KUKA KRL program: EPS_2_25694_SR01_A_NEW_20251202031151.src

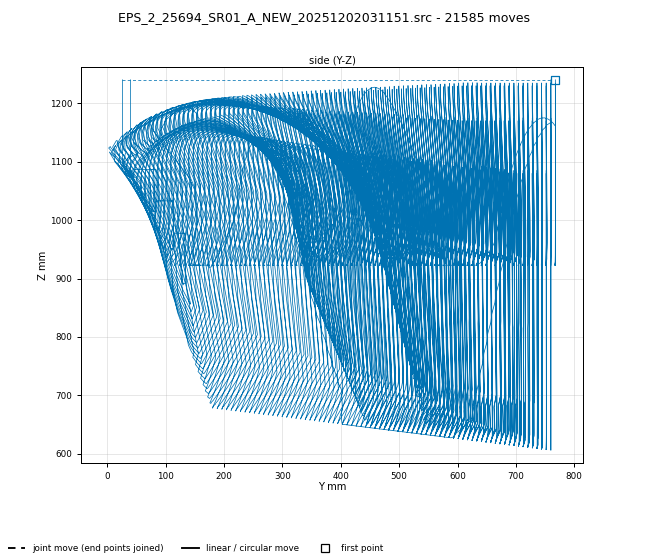
[picture p0: tool path of EPS_2_25694_SR01_A_NEW_20251202031151.src, 21585 of 21587 moves have a stored position in this frame; points joined in program order, loops and branches not executed]
&ACCESS RVP
&REL 4
&COMMENT QRS 19112012
&PARAM EDITMASK = *
DEF PART()
EXT BAS (BAS_COMMAND :IN,REAL :IN )
INT I
BAS (#INITMOV,0 )

;KUKA QRS Post kuka4.cps  Date:22-06-2017 !

File_ID=2935

QRS_PRE_INIT()

;Init var - Until changes are made in qrs_pre_init
Outlet_Square_prg=0
Inlet_1_Square_prg=0
Inlet_2_Square_prg=0
Inlet_3_Square_prg=0
Inlet_4_Square_prg=0
Inlet_5_Square_prg=0

Outlet_1={X 0.000, Y 612.000, Z 964.000, B 0.000, E1 0.000 }
Inlet_1={X 0.000, Y 612.000, Z 904.000, B 0.000, E1 90.000 }
Inlet_2={X 0.000, Y 692.870, Z 705.000, B 0.000, E1 260.000 }
Outlet_1_type=533
Inlet_1_type=533
Inlet_2_type=251
;QRS#1=Sidecore dimensions
;QRS#2=525-21" Concrete
;QRS#3=525-21" Concrete
;QRS#4=250-10" PVC SDR 35
;QRS#5=
;QRS#6=
;QRS#7=
;QRS#8=
;QRS#9=S306-32
;QRS#10=S306-32
;QRS#11=14M PSX
;QRS#12=
;QRS#13=
;QRS#14=
;QRS#15=
;QRS#16=1524x152x1676 5,5'
;QRS#17=EPS Height
;QRS#18=1230,5
;QRS#19=*
;QRS#20= UPDATED VERSION 22-06-2017
;QRS#21=*
Outlet_Square=0350
Inlet_1_Square=0350
Inlet_2_Square=0100
Inlet_3_Square=0
Inlet_4_Square=0
Inlet_5_Square=0
Mill_Square=1
Outlet_Square_Prg=263
Inlet_1_Square_prg=263
Inlet_2_Square_prg=205

QRS_INIT()

$ADVANCE=5

; T1
PTP {E1 173.088,E2 173.088}
PTP {X 0,Y 767.616,A -85,B 0,C 180,E1 173.088,E2 173.088,E3 0,E4 0,E5 0,E6 0}
QRS_SPEED_INIT()
LIN {X 0,Y 767.616,Z 1240.5,A -85,B 0,C 180,E1 173.088,E2 173.088,E3 0,E4 0,E5 0,E6 0} C_VEL
LIN {X 0,Y 767.616,Z 1171.13,A -85,B 0,C 180,E1 173.088,E2 173.088} C_VEL
LIN {X 0,Y 767.616,Z 1163.237,A -85,B 0,C 180,E1 173.088,E2 173.088} C_VEL
LIN {X 0,Y 767.6,Z 1161.315,A -85,B 0,C 180,E1 173.278,E2 173.278} C_VEL
LIN {X 0,Y 767.645,Z 1164.897,A -85,B 0,C 180,E1 174.209,E2 174.209} C_VEL
LIN {X 0,Y 767.804,Z 1167.383,A -85,B 0,C 180,E1 174.959,E2 174.959} C_VEL
LIN {X 0,Y 767.62,Z 1170.432,A -85,B 0,C 180,E1 176.081,E2 176.081} C_VEL
LIN {X 0,Y 767.646,Z 1172.644,A -85,B 0,C 180,E1 177.202,E2 177.202} C_VEL
LIN {X 0,Y 767.795,Z 1174.074,A -85,B 0,C 180,E1 178.323,E2 178.323} C_VEL
LIN {X 0,Y 767.585,Z 1174.722,A -85,B 0,C 180,E1 179.069,E2 179.069} C_VEL
LIN {X 0,Y 767.644,Z 1174.677,A -85,B 0,C 180,E1 180.934,E2 180.934} C_VEL
LIN {X 0,Y 767.742,Z 1173.598,A -85,B 0,C 180,E1 182.054,E2 182.054} C_VEL
LIN {X 0,Y 767.614,Z 1172.514,A -85,B 0,C 180,E1 182.801,E2 182.801} C_VEL
LIN {X 0,Y 767.666,Z 1170.222,A -85,B 0,C 180,E1 183.922,E2 183.922} C_VEL
LIN {X 0,Y 767.825,Z 1168.163,A -85,B 0,C 180,E1 184.669,E2 184.669} C_VEL
LIN {X 0,Y 767.693,Z 1165.832,A -85,B 0,C 180,E1 185.419,E2 185.419} C_VEL
LIN {X 0,Y 767.64,Z 1163.158,A -85,B 0,C 180,E1 186.17,E2 186.17} C_VEL
LIN {X 0,Y 767.709,Z 1160.308,A -85,B 0,C 180,E1 186.878,E2 186.878} C_VEL
LIN {X 0,Y 767.81,Z 1156.374,A -85,B 0,C 180,E1 187.718,E2 187.718} C_VEL
LIN {X 0,Y 767.635,Z 1150.131,A -85,B 0,C 180,E1 188.898,E2 188.898} C_VEL
LIN {X 0,Y 767.742,Z 1144.316,A -85,B 0,C 180,E1 189.842,E2 189.842} C_VEL
LIN {X 0,Y 767.829,Z 1139.474,A -85,B 0,C 180,E1 190.552,E2 190.552} C_VEL
LIN {X 0,Y 767.685,Z 1132.395,A -85,B 0,C 180,E1 191.504,E2 191.504} C_VEL
LIN {X 0,Y 767.755,Z 1123.331,A -85,B 0,C 180,E1 192.576,E2 192.576} C_VEL
LIN {X 0,Y 767.785,Z 1116.439,A -85,B 0,C 180,E1 193.319,E2 193.319} C_VEL
LIN {X 0,Y 767.704,Z 1107.11,A -85,B 0,C 180,E1 194.231,E2 194.231} C_VEL
LIN {X 0,Y 767.763,Z 1099.606,A -85,B 0,C 180,E1 194.904,E2 194.904} C_VEL
LIN {X 0,Y 767.79,Z 1090.202,A -85,B 0,C 180,E1 195.677,E2 195.677} C_VEL
LIN {X 0,Y 767.737,Z 1080.825,A -85,B 0,C 180,E1 196.385,E2 196.385} C_VEL
LIN {X 0,Y 767.747,Z 1071.416,A -85,B 0,C 180,E1 197.039,E2 197.039} C_VEL
LIN {X 0,Y 767.76,Z 1060.856,A -85,B 0,C 180,E1 197.71,E2 197.71} C_VEL
LIN {X 0,Y 767.758,Z 1050.335,A -85,B 0,C 180,E1 198.323,E2 198.323} C_VEL
LIN {X 0,Y 767.76,Z 1039.977,A -85,B 0,C 180,E1 198.877,E2 198.877} C_VEL
LIN {X 0,Y 767.736,Z 1028.552,A -85,B 0,C 180,E1 199.433,E2 199.433} C_VEL
LIN {X 0,Y 767.781,Z 1015.782,A -85,B 0,C 180,E1 199.989,E2 199.989} C_VEL
LIN {X 0,Y 767.752,Z 1003.711,A -85,B 0,C 180,E1 200.462,E2 200.462} C_VEL
LIN {X 0,Y 767.714,Z 992.2,A -85,B 0,C 180,E1 200.866,E2 200.866} C_VEL
LIN {X 0,Y 767.776,Z 978.277,A -85,B 0,C 180,E1 201.291,E2 201.291} C_VEL
LIN {X 0,Y 767.685,Z 965.195,A -85,B 0,C 180,E1 201.639,E2 201.639} C_VEL
LIN {X 0,Y 767.732,Z 952.435,A -85,B 0,C 180,E1 201.925,E2 201.925} C_VEL
LIN {X 0,Y 767.714,Z 939.22,A -85,B 0,C 180,E1 202.172,E2 202.172} C_VEL
LIN {X 0,Y 767.488,Z 929.301,A -85,B 0,C 180,E1 202.333,E2 202.333} C_VEL
LIN {X 0,Y 766.705,Z 923.03,A -85,B 0,C 180,E1 202.439,E2 202.439} C_VEL
LIN {X 0,Y 767.325,Z 923.03,A -85,B 0,C 180,E1 202.504,E2 202.504} C_VEL
LIN {X 0,Y 767.822,Z 923.03,A -85,B 0,C 180,E1 202.614,E2 202.614} C_VEL
LIN {X 0,Y 767.644,Z 923.03,A -85,B 0,C 180,E1 203.63,E2 203.63} C_VEL
LIN {X 0,Y 767.743,Z 923.03,A -85,B 0,C 180,E1 208.169,E2 208.169} C_VEL
LIN {X 0,Y 767.312,Z 923.03,A -85,B 0,C 180,E1 210.325,E2 210.325} C_VEL
LIN {X 0,Y 767.713,Z 923.03,A -85,B 0,C 180,E1 212.493,E2 212.493} C_VEL
LIN {X 0,Y 767.395,Z 923.03,A -85,B 0,C 180,E1 213.845,E2 213.845} C_VEL
LIN {X 0,Y 767.696,Z 923.03,A -85,B 0,C 180,E1 217.093,E2 217.093} C_VEL
LIN {X 0,Y 767.102,Z 923.03,A -85,B 0,C 180,E1 220.031,E2 220.031} C_VEL
LIN {X 0,Y 767.566,Z 923.03,A -85,B 0,C 180,E1 221.878,E2 221.878} C_VEL
LIN {X 0,Y 767.622,Z 923.03,A -85,B 0,C 180,E1 222.894,E2 222.894} C_VEL
LIN {X 0,Y 767.591,Z 923.03,A -85,B 0,C 180,E1 227.109,E2 227.109} C_VEL
LIN {X 0,Y 767.541,Z 923.03,A -85,B 0,C 180,E1 228.12,E2 228.12} C_VEL
LIN {X 0,Y 767.131,Z 923.03,A -85,B 0,C 180,E1 230.554,E2 230.554} C_VEL
LIN {X 0,Y 767.736,Z 923.03,A -85,B 0,C 180,E1 232.966,E2 232.966} C_VEL
LIN {X 0,Y 767.601,Z 923.03,A -85,B 0,C 180,E1 236.132,E2 236.132} C_VEL
LIN {X 0,Y 767.507,Z 923.03,A -85,B 0,C 180,E1 237.497,E2 237.497} C_VEL
LIN {X 0,Y 767.223,Z 923.03,A -85,B 0,C 180,E1 239.69,E2 239.69} C_VEL
LIN {X 0,Y 767.749,Z 923.03,A -85,B 0,C 180,E1 241.832,E2 241.832} C_VEL
LIN {X 0,Y 767.82,Z 923.03,A -85,B 0,C 180,E1 246.871,E2 246.871} C_VEL
LIN {X 0,Y 767.647,Z 923.03,A -85,B 0,C 180,E1 246.92,E2 246.92} C_VEL
LIN {X 0,Y 767.578,Z 923.795,A -85,B 0,C 180,E1 246.945,E2 246.945} C_VEL
LIN {X 0,Y 767.629,Z 977.672,A -85,B 0,C 180,E1 247.486,E2 247.486} C_VEL
LIN {X 0,Y 767.739,Z 990.959,A -85,B 0,C 180,E1 247.656,E2 247.656} C_VEL
LIN {X 0,Y 767.675,Z 1003.622,A -85,B 0,C 180,E1 247.858,E2 247.858} C_VEL
LIN {X 0,Y 767.717,Z 1014.508,A -85,B 0,C 180,E1 248.07,E2 248.07} C_VEL
LIN {X 0,Y 767.776,Z 1030.265,A -85,B 0,C 180,E1 248.446,E2 248.446} C_VEL
LIN {X 0,Y 767.72,Z 1042.52,A -85,B 0,C 180,E1 248.785,E2 248.785} C_VEL
LIN {X 0,Y 767.741,Z 1055.126,A -85,B 0,C 180,E1 249.188,E2 249.188} C_VEL
LIN {X 0,Y 767.772,Z 1067.885,A -85,B 0,C 180,E1 249.651,E2 249.651} C_VEL
LIN {X 0,Y 767.73,Z 1079.832,A -85,B 0,C 180,E1 250.134,E2 250.134} C_VEL
LIN {X 0,Y 767.776,Z 1092.122,A -85,B 0,C 180,E1 250.692,E2 250.692} C_VEL
LIN {X 0,Y 767.784,Z 1103.222,A -85,B 0,C 180,E1 251.247,E2 251.247} C_VEL
LIN {X 0,Y 767.77,Z 1114.39,A -85,B 0,C 180,E1 251.862,E2 251.862} C_VEL
LIN {X 0,Y 767.759,Z 1124.576,A -85,B 0,C 180,E1 252.474,E2 252.474} C_VEL
LIN {X 0,Y 767.741,Z 1133.933,A -85,B 0,C 180,E1 253.083,E2 253.083} C_VEL
LIN {X 0,Y 767.808,Z 1144.001,A -85,B 0,C 180,E1 253.803,E2 253.803} C_VEL
LIN {X 0,Y 767.769,Z 1153.202,A -85,B 0,C 180,E1 254.517,E2 254.517} C_VEL
LIN {X 0,Y 767.702,Z 1162.313,A -85,B 0,C 180,E1 255.288,E2 255.288} C_VEL
LIN {X 0,Y 767.775,Z 1170.487,A -85,B 0,C 180,E1 256.045,E2 256.045} C_VEL
LIN {X 0,Y 767.79,Z 1178.25,A -85,B 0,C 180,E1 256.827,E2 256.827} C_VEL
LIN {X 0,Y 767.68,Z 1185.844,A -85,B 0,C 180,E1 257.662,E2 257.662} C_VEL
LIN {X 0,Y 767.726,Z 1192.732,A -85,B 0,C 180,E1 258.497,E2 258.497} C_VEL
LIN {X 0,Y 767.83,Z 1198.109,A -85,B 0,C 180,E1 259.211,E2 259.211} C_VEL
LIN {X 0,Y 767.639,Z 1204.639,A -85,B 0,C 180,E1 260.157,E2 260.157} C_VEL
LIN {X 0,Y 767.667,Z 1210.401,A -85,B 0,C 180,E1 261.102,E2 261.102} C_VEL
LIN {X 0,Y 767.825,Z 1215.453,A -85,B 0,C 180,E1 262.047,E2 262.047} C_VEL
LIN {X 0,Y 767.632,Z 1221.05,A -85,B 0,C 180,E1 263.258,E2 263.258} C_VEL
LIN {X 0,Y 767.708,Z 1224.727,A -85,B 0,C 180,E1 264.206,E2 264.206} C_VEL
LIN {X 0,Y 767.823,Z 1227.22,A -85,B 0,C 180,E1 264.957,E2 264.957} C_VEL
LIN {X 0,Y 767.655,Z 1229.333,A -85,B 0,C 180,E1 265.704,E2 265.704} C_VEL
LIN {X 0,Y 767.605,Z 1231.115,A -85,B 0,C 180,E1 266.452,E2 266.452} C_VEL
LIN {X 0,Y 767.683,Z 1232.567,A -85,B 0,C 180,E1 267.2,E2 267.2} C_VEL
LIN {X 0,Y 767.835,Z 1233.648,A -85,B 0,C 180,E1 267.947,E2 267.947} C_VEL
LIN {X 0,Y 767.616,Z 1234.703,A -85,B 0,C 180,E1 269.066,E2 269.066} C_VEL
LIN {X 0,Y 767.835,Z 1234.661,A -85,B 0,C 180,E1 270.931,E2 270.931} C_VEL
LIN {X 0,Y 767.781,Z 1234.037,A -85,B 0,C 180,E1 271.678,E2 271.678} C_VEL
LIN {X 0,Y 767.801,Z 1232.548,A -85,B 0,C 180,E1 272.798,E2 272.798} C_VEL
LIN {X 0,Y 767.672,Z 1231.107,A -85,B 0,C 180,E1 273.545,E2 273.545} C_VEL
LIN {X 0,Y 767.7,Z 1228.315,A -85,B 0,C 180,E1 274.667,E2 274.667} C_VEL
LIN {X 0,Y 767.838,Z 1225.965,A -85,B 0,C 180,E1 275.415,E2 275.415} C_VEL
LIN {X 0,Y 767.7,Z 1223.339,A -85,B 0,C 180,E1 276.166,E2 276.166} C_VEL
LIN {X 0,Y 767.635,Z 1220.661,A -85,B 0,C 180,E1 276.839,E2 276.839} C_VEL
LIN {X 0,Y 767.801,Z 1215.469,A -85,B 0,C 180,E1 277.951,E2 277.951} C_VEL
LIN {X 0,Y 767.723,Z 1210.407,A -85,B 0,C 180,E1 278.895,E2 278.895} C_VEL
LIN {X 0,Y 767.638,Z 1204.655,A -85,B 0,C 180,E1 279.841,E2 279.841} C_VEL
LIN {X 0,Y 767.786,Z 1198.133,A -85,B 0,C 180,E1 280.787,E2 280.787} C_VEL
LIN {X 0,Y 767.73,Z 1190.839,A -85,B 0,C 180,E1 281.739,E2 281.739} C_VEL
LIN {X 0,Y 767.66,Z 1183.778,A -85,B 0,C 180,E1 282.575,E2 282.575} C_VEL
LIN {X 0,Y 767.78,Z 1175.272,A -85,B 0,C 180,E1 283.479,E2 283.479} C_VEL
LIN {X 0,Y 767.762,Z 1167.631,A -85,B 0,C 180,E1 284.227,E2 284.227} C_VEL
LIN {X 0,Y 767.71,Z 1159.021,A -85,B 0,C 180,E1 284.999,E2 284.999} C_VEL
LIN {X 0,Y 767.753,Z 1150.824,A -85,B 0,C 180,E1 285.675,E2 285.675} C_VEL
LIN {X 0,Y 767.789,Z 1141.234,A -85,B 0,C 180,E1 286.4,E2 286.4} C_VEL
LIN {X 0,Y 767.753,Z 1132.152,A -85,B 0,C 180,E1 287.036,E2 287.036} C_VEL
LIN {X 0,Y 767.756,Z 1120.627,A -85,B 0,C 180,E1 287.769,E2 287.769} C_VEL
LIN {X 0,Y 767.748,Z 1110.08,A -85,B 0,C 180,E1 288.382,E2 288.382} C_VEL
LIN {X 0,Y 767.777,Z 1099.692,A -85,B 0,C 180,E1 288.935,E2 288.935} C_VEL
LIN {X 0,Y 767.775,Z 1088.232,A -85,B 0,C 180,E1 289.491,E2 289.491} C_VEL
LIN {X 0,Y 767.732,Z 1076.974,A -85,B 0,C 180,E1 289.987,E2 289.987} C_VEL
LIN {X 0,Y 767.792,Z 1064.346,A -85,B 0,C 180,E1 290.483,E2 290.483} C_VEL
LIN {X 0,Y 767.771,Z 1051.74,A -85,B 0,C 180,E1 290.924,E2 290.924} C_VEL
LIN {X 0,Y 767.668,Z 1038.39,A -85,B 0,C 180,E1 291.336,E2 291.336} C_VEL
LIN {X 0,Y 767.771,Z 1025.24,A -85,B 0,C 180,E1 291.68,E2 291.68} C_VEL
LIN {X 0,Y 767.797,Z 1012.208,A -85,B 0,C 180,E1 291.972,E2 291.972} C_VEL
LIN {X 0,Y 767.692,Z 999.283,A -85,B 0,C 180,E1 292.216,E2 292.216} C_VEL
LIN {X 0,Y 767.662,Z 989.615,A -85,B 0,C 180,E1 292.367,E2 292.367} C_VEL
LIN {X 0,Y 767.711,Z 970.479,A -85,B 0,C 180,E1 292.587,E2 292.587} C_VEL
LIN {X 0,Y 767.567,Z 923.965,A -85,B 0,C 180,E1 293.054,E2 293.054} C_VEL
LIN {X 0,Y 767.609,Z 923.03,A -85,B 0,C 180,E1 293.072,E2 293.072} C_VEL
LIN {X 0,Y 767.756,Z 923.03,A -85,B 0,C 180,E1 293.108,E2 293.108} C_VEL
LIN {X 0,Y 767.439,Z 923.03,A -85,B 0,C 180,E1 294.021,E2 294.021} C_VEL
LIN {X 0,Y 767.75,Z 923.03,A -85,B 0,C 180,E1 298.166,E2 298.166} C_VEL
LIN {X 0,Y 767.337,Z 923.03,A -85,B 0,C 180,E1 300.324,E2 300.324} C_VEL
LIN {X 0,Y 767.758,Z 923.03,A -85,B 0,C 180,E1 302.488,E2 302.488} C_VEL
LIN {X 0,Y 767.431,Z 923.03,A -85,B 0,C 180,E1 303.849,E2 303.849} C_VEL
LIN {X 0,Y 767.734,Z 923.03,A -85,B 0,C 180,E1 307.096,E2 307.096} C_VEL
LIN {X 0,Y 767.112,Z 923.03,A -85,B 0,C 180,E1 310.032,E2 310.032} C_VEL
LIN {X 0,Y 767.566,Z 923.03,A -85,B 0,C 180,E1 311.875,E2 311.875} C_VEL
LIN {X 0,Y 767.634,Z 923.03,A -85,B 0,C 180,E1 312.895,E2 312.895} C_VEL
LIN {X 0,Y 767.633,Z 923.03,A -85,B 0,C 180,E1 317.102,E2 317.102} C_VEL
LIN {X 0,Y 767.581,Z 923.03,A -85,B 0,C 180,E1 318.123,E2 318.123} C_VEL
LIN {X 0,Y 767.123,Z 923.03,A -85,B 0,C 180,E1 320.554,E2 320.554} C_VEL
LIN {X 0,Y 767.7,Z 923.03,A -85,B 0,C 180,E1 322.964,E2 322.964} C_VEL
LIN {X 0,Y 767.576,Z 923.03,A -85,B 0,C 180,E1 326.13,E2 326.13} C_VEL
LIN {X 0,Y 767.481,Z 923.03,A -85,B 0,C 180,E1 327.496,E2 327.496} C_VEL
LIN {X 0,Y 767.213,Z 923.03,A -85,B 0,C 180,E1 329.687,E2 329.687} C_VEL
LIN {X 0,Y 767.767,Z 923.03,A -85,B 0,C 180,E1 331.832,E2 331.832} C_VEL
LIN {X 0,Y 767.786,Z 923.03,A -85,B 0,C 180,E1 335.988,E2 335.988} C_VEL
LIN {X 0,Y 767.774,Z 923.03,A -85,B 0,C 180,E1 340.011,E2 340.011} C_VEL
LIN {X 0,Y 767.215,Z 923.03,A -85,B 0,C 180,E1 343.947,E2 343.947} C_VEL
LIN {X 0,Y 767.659,Z 923.03,A -85,B 0,C 180,E1 345.865,E2 345.865} C_VEL
LIN {X 0,Y 767.793,Z 923.03,A -85,B 0,C 180,E1 349.685,E2 349.685} C_VEL
LIN {X 0,Y 767.822,Z 923.03,A -85,B 0,C 180,E1 353.457,E2 353.457} C_VEL
LIN {X 0,Y 767.841,Z 923.03,A -85,B 0,C 180,E1 357.918,E2 357.918} C_VEL
LIN {X 0,Y 767.412,Z 923.03,A -85,B 0,C 180,E1 358.035,E2 358.035} C_VEL
LIN {X 0,Y 766.897,Z 923.03,A -85,B 0,C 180,E1 358.098,E2 358.098} C_VEL
LIN {X 0,Y 767.682,Z 928.435,A -85,B 0,C 180,E1 358.165,E2 358.165} C_VEL
LIN {X 0,Y 767.803,Z 954.739,A -85,B 0,C 180,E1 358.423,E2 358.423} C_VEL
LIN {X 0,Y 767.86,Z 965.313,A -85,B 0,C 180,E1 358.583,E2 358.583} C_VEL
LIN {X 0,Y 767.858,Z 973.85,A -85,B 0,C 180,E1 358.755,E2 358.755} C_VEL
LIN {X 0,Y 767.845,Z 982.97,A -85,B 0,C 180,E1 358.98,E2 358.98} C_VEL
LIN {X 0,Y 767.836,Z 991.896,A -85,B 0,C 180,E1 359.253,E2 359.253} C_VEL
LIN {X 0,Y 767.828,Z 999.738,A -85,B 0,C 180,E1 359.532,E2 359.532} C_VEL
LIN {X 0,Y 767.806,Z 1008.817,A -85,B 0,C 180,E1 359.905,E2 359.905} C_VEL
LIN {X 0,Y 767.817,Z 1016.57,A -85,B 0,C 180,E1 360.278,E2 360.278} C_VEL
LIN {X 0,Y 767.843,Z 1023.443,A -85,B 0,C 180,E1 360.651,E2 360.651} C_VEL
LIN {X 0,Y 767.856,Z 1031.11,A -85,B 0,C 180,E1 361.118,E2 361.118} C_VEL
LIN {X 0,Y 767.816,Z 1037.833,A -85,B 0,C 180,E1 361.584,E2 361.584} C_VEL
LIN {X 0,Y 767.828,Z 1046.128,A -85,B 0,C 180,E1 362.237,E2 362.237} C_VEL
LIN {X 0,Y 767.834,Z 1052.24,A -85,B 0,C 180,E1 362.797,E2 362.797} C_VEL
LIN {X 0,Y 767.79,Z 1057.697,A -85,B 0,C 180,E1 363.358,E2 363.358} C_VEL
LIN {X 0,Y 767.808,Z 1062.52,A -85,B 0,C 180,E1 363.918,E2 363.918} C_VEL
LIN {X 0,Y 767.858,Z 1066.717,A -85,B 0,C 180,E1 364.479,E2 364.479} C_VEL
LIN {X 0,Y 767.776,Z 1070.444,A -85,B 0,C 180,E1 365.041,E2 365.041} C_VEL
LIN {X 0,Y 767.747,Z 1073.688,A -85,B 0,C 180,E1 365.603,E2 365.603} C_VEL
LIN {X 0,Y 767.808,Z 1076.465,A -85,B 0,C 180,E1 366.165,E2 366.165} C_VEL
LIN {X 0,Y 767.817,Z 1079.418,A -85,B 0,C 180,E1 366.877,E2 366.877} C_VEL
LIN {X 0,Y 767.756,Z 1081.384,A -85,B 0,C 180,E1 367.481,E2 367.481} C_VEL
LIN {X 0,Y 767.762,Z 1082.621,A -85,B 0,C 180,E1 367.951,E2 367.951} C_VEL
LIN {X 0,Y 767.82,Z 1083.578,A -85,B 0,C 180,E1 368.422,E2 368.422} C_VEL
LIN {X 0,Y 767.773,Z 1084.727,A -85,B 0,C 180,E1 369.366,E2 369.366} C_VEL
LIN {X 0,Y 767.751,Z 1084.916,A -85,B 0,C 180,E1 369.839,E2 369.839} C_VEL
LIN {X 0,Y 767.782,Z 1084.839,A -85,B 0,C 180,E1 370.312,E2 370.312} C_VEL
LIN {X 0,Y 767.852,Z 1084.497,A -85,B 0,C 180,E1 370.786,E2 370.786} C_VEL
LIN {X 0,Y 767.8,Z 1083.921,A -85,B 0,C 180,E1 371.262,E2 371.262} C_VEL
LIN {X 0,Y 767.746,Z 1083.082,A -85,B 0,C 180,E1 371.738,E2 371.738} C_VEL
LIN {X 0,Y 767.744,Z 1081.966,A -85,B 0,C 180,E1 372.215,E2 372.215} C_VEL
LIN {X 0,Y 767.795,Z 1080.566,A -85,B 0,C 180,E1 372.692,E2 372.692} C_VEL
LIN {X 0,Y 767.787,Z 1077.674,A -85,B 0,C 180,E1 373.474,E2 373.474} C_VEL
LIN {X 0,Y 767.765,Z 1074.632,A -85,B 0,C 180,E1 374.13,E2 374.13} C_VEL
LIN {X 0,Y 767.803,Z 1071.423,A -85,B 0,C 180,E1 374.707,E2 374.707} C_VEL
LIN {X 0,Y 767.831,Z 1067.715,A -85,B 0,C 180,E1 375.286,E2 375.286} C_VEL
LIN {X 0,Y 767.772,Z 1063.48,A -85,B 0,C 180,E1 375.868,E2 375.868} C_VEL
LIN {X 0,Y 767.817,Z 1057.741,A -85,B 0,C 180,E1 376.547,E2 376.547} C_VEL
LIN {X 0,Y 767.845,Z 1051.803,A -85,B 0,C 180,E1 377.155,E2 377.155} C_VEL
LIN {X 0,Y 767.798,Z 1044.974,A -85,B 0,C 180,E1 377.767,E2 377.767} C_VEL
LIN {X 0,Y 767.836,Z 1037.134,A -85,B 0,C 180,E1 378.379,E2 378.379} C_VEL
LIN {X 0,Y 767.851,Z 1029.859,A -85,B 0,C 180,E1 378.871,E2 378.871} C_VEL
LIN {X 0,Y 767.826,Z 1022.668,A -85,B 0,C 180,E1 379.303,E2 379.303} C_VEL
LIN {X 0,Y 767.83,Z 1014.515,A -85,B 0,C 180,E1 379.736,E2 379.736} C_VEL
LIN {X 0,Y 767.84,Z 1006.03,A -85,B 0,C 180,E1 380.123,E2 380.123} C_VEL
LIN {X 0,Y 767.833,Z 997.385,A -85,B 0,C 180,E1 380.467,E2 380.467} C_VEL
LIN {X 0,Y 767.802,Z 988.868,A -85,B 0,C 180,E1 380.756,E2 380.756} C_VEL
LIN {X 0,Y 767.856,Z 979.688,A -85,B 0,C 180,E1 381.014,E2 381.014} C_VEL
LIN {X 0,Y 767.86,Z 969.785,A -85,B 0,C 180,E1 381.244,E2 381.244} C_VEL
LIN {X 0,Y 767.815,Z 959.779,A -85,B 0,C 180,E1 381.417,E2 381.417} C_VEL
LIN {X 0,Y 767.834,Z 950.7,A -85,B 0,C 180,E1 381.532,E2 381.532} C_VEL
LIN {X 0,Y 767.761,Z 926.079,A -85,B 0,C 180,E1 381.766,E2 381.766} C_VEL
LIN {X 0,Y 766.941,Z 923.622,A -85,B 0,C 180,E1 381.802,E2 381.802} C_VEL
LIN {X 0,Y 766.65,Z 923.03,A -85,B 0,C 180,E1 381.819,E2 381.819} C_VEL
LIN {X 0,Y 767.601,Z 923.03,A -85,B 0,C 180,E1 381.989,E2 381.989} C_VEL
LIN {X 0,Y 767.531,Z 923.03,A -85,B 0,C 180,E1 384.018,E2 384.018} C_VEL
LIN {X 0,Y 767.633,Z 923.03,A -85,B 0,C 180,E1 386.074,E2 386.074} C_VEL
LIN {X 0,Y 767.775,Z 923.03,A -85,B 0,C 180,E1 390.385,E2 390.385} C_VEL
LIN {X 0,Y 767.726,Z 923.03,A -85,B 0,C 180,E1 394.729,E2 394.729} C_VEL
LIN {X 0,Y 767.234,Z 923.03,A -85,B 0,C 180,E1 397.059,E2 397.059} C_VEL
LIN {X 0,Y 767.688,Z 923.03,A -85,B 0,C 180,E1 399.408,E2 399.408} C_VEL
LIN {X 0,Y 767.67,Z 923.03,A -85,B 0,C 180,E1 400.085,E2 400.085} C_VEL
LIN {X 0,Y 767.475,Z 923.03,A -85,B 0,C 180,E1 404.439,E2 404.439} C_VEL
LIN {X 0,Y 767.642,Z 923.03,A -85,B 0,C 180,E1 405.573,E2 405.573} C_VEL
LIN {X 0,Y 767.693,Z 923.03,A -85,B 0,C 180,E1 409.912,E2 409.912} C_VEL
LIN {X 0,Y 767.697,Z 923.03,A -85,B 0,C 180,E1 410.592,E2 410.592} C_VEL
LIN {X 0,Y 767.21,Z 923.03,A -85,B 0,C 180,E1 412.951,E2 412.951} C_VEL
LIN {X 0,Y 767.666,Z 923.03,A -85,B 0,C 180,E1 415.267,E2 415.267} C_VEL
LIN {X 0,Y 767.73,Z 923.03,A -85,B 0,C 180,E1 419.62,E2 419.62} C_VEL
LIN {X 0,Y 767.786,Z 923.03,A -85,B 0,C 180,E1 423.531,E2 423.531} C_VEL
LIN {X 0,Y 767.789,Z 923.03,A -85,B 0,C 180,E1 423.932,E2 423.932} C_VEL
LIN {X 0,Y 767.77,Z 923.03,A -85,B 0,C 180,E1 428.016,E2 428.016} C_VEL
LIN {X 0,Y 767.757,Z 923.03,A -85,B 0,C 180,E1 431.986,E2 431.986} C_VEL
LIN {X 0,Y 767.458,Z 923.03,A -85,B 0,C 180,E1 433.931,E2 433.931} C_VEL
LIN {X 0,Y 767.591,Z 923.03,A -85,B 0,C 180,E1 435.866,E2 435.866} C_VEL
LIN {X 0,Y 767.792,Z 923.03,A -85,B 0,C 180,E1 439.687,E2 439.687} C_VEL
LIN {X 0,Y 767.847,Z 923.03,A -85,B 0,C 180,E1 443.459,E2 443.459} C_VEL
LIN {X 0,Y 767.872,Z 923.03,A -85,B 0,C 180,E1 447.203,E2 447.203} C_VEL
LIN {X 0,Y 767.868,Z 923.03,A -85,B 0,C 180,E1 450.934,E2 450.934} C_VEL
LIN {X 0,Y 767.84,Z 923.03,A -85,B 0,C 180,E1 454.669,E2 454.669} C_VEL
LIN {X 0,Y 767.829,Z 923.03,A -85,B 0,C 180,E1 458.424,E2 458.424} C_VEL
LIN {X 0,Y 767.822,Z 923.03,A -85,B 0,C 180,E1 462.216,E2 462.216} C_VEL
LIN {X 0,Y 767.858,Z 923.03,A -85,B 0,C 180,E1 466.221,E2 466.221} C_VEL
LIN {X 0,Y 767.739,Z 923.03,A -85,B 0,C 180,E1 469.989,E2 469.989} C_VEL
LIN {X 0,Y 767.734,Z 923.03,A -85,B 0,C 180,E1 474.014,E2 474.014} C_VEL
LIN {X 0,Y 767.335,Z 923.03,A -85,B 0,C 180,E1 476.401,E2 476.401} C_VEL
LIN {X 0,Y 767.741,Z 923.03,A -85,B 0,C 180,E1 478.168,E2 478.168} C_VEL
LIN {X 0,Y 767.316,Z 923.03,A -85,B 0,C 180,E1 480.328,E2 480.328} C_VEL
LIN {X 0,Y 767.737,Z 923.03,A -85,B 0,C 180,E1 482.492,E2 482.492} C_VEL
LIN {X 0,Y 767.415,Z 923.03,A -85,B 0,C 180,E1 483.853,E2 483.853} C_VEL
LIN {X 0,Y 767.681,Z 923.03,A -85,B 0,C 180,E1 487.096,E2 487.096} C_VEL
LIN {X 0,Y 767.162,Z 923.03,A -85,B 0,C 180,E1 490.041,E2 490.041} C_VEL
LIN {X 0,Y 767.682,Z 923.03,A -85,B 0,C 180,E1 491.87,E2 491.87} C_VEL
LIN {X 0,Y 767.693,Z 923.03,A -85,B 0,C 180,E1 492.904,E2 492.904} C_VEL
LIN {X 0,Y 767.672,Z 923.03,A -85,B 0,C 180,E1 494.428,E2 494.428} C_VEL
LIN {X 0,Y 767.629,Z 923.03,A -85,B 0,C 180,E1 495.573,E2 495.573} C_VEL
LIN {X 0,Y 767.694,Z 923.03,A -85,B 0,C 180,E1 499.916,E2 499.916} C_VEL
LIN {X 0,Y 767.699,Z 923.03,A -85,B 0,C 180,E1 500.593,E2 500.593} C_VEL
LIN {X 0,Y 767.207,Z 923.03,A -85,B 0,C 180,E1 502.956,E2 502.956} C_VEL
LIN {X 0,Y 767.69,Z 923.03,A -85,B 0,C 180,E1 505.269,E2 505.269} C_VEL
LIN {X 0,Y 767.733,Z 923.03,A -85,B 0,C 180,E1 509.625,E2 509.625} C_VEL
LIN {X 0,Y 767.776,Z 923.03,A -85,B 0,C 180,E1 513.539,E2 513.539} C_VEL
LIN {X 0,Y 767.785,Z 923.03,A -85,B 0,C 180,E1 513.932,E2 513.932} C_VEL
LIN {X 0,Y 767.701,Z 923.03,A -85,B 0,C 180,E1 516.902,E2 516.902} C_VEL
LIN {X 0,Y 767.753,Z 923.03,A -85,B 0,C 180,E1 517.407,E2 517.407} C_VEL
LIN {X 0,Y 767.323,Z 923.03,A -85,B 0,C 180,E1 517.489,E2 517.489} C_VEL
LIN {X 0,Y 767.582,Z 936.224,A -85,B 0,C 180,E1 517.688,E2 517.688} C_VEL
LIN {X 0,Y 767.747,Z 945.654,A -85,B 0,C 180,E1 517.854,E2 517.854} C_VEL
LIN {X 0,Y 767.798,Z 957.639,A -85,B 0,C 180,E1 518.099,E2 518.099} C_VEL
LIN {X 0,Y 767.761,Z 969.731,A -85,B 0,C 180,E1 518.386,E2 518.386} C_VEL
LIN {X 0,Y 767.673,Z 980.092,A -85,B 0,C 180,E1 518.666,E2 518.666} C_VEL
LIN {X 0,Y 767.749,Z 995.086,A -85,B 0,C 180,E1 519.141,E2 519.141} C_VEL
LIN {X 0,Y 767.699,Z 1008.532,A -85,B 0,C 180,E1 519.629,E2 519.629} C_VEL
LIN {X 0,Y 767.775,Z 1019.516,A -85,B 0,C 180,E1 520.076,E2 520.076} C_VEL
LIN {X 0,Y 767.782,Z 1031.84,A -85,B 0,C 180,E1 520.634,E2 520.634} C_VEL
LIN {X 0,Y 767.731,Z 1042.97,A -85,B 0,C 180,E1 521.187,E2 521.187} C_VEL
LIN {X 0,Y 767.771,Z 1054.163,A -85,B 0,C 180,E1 521.803,E2 521.803} C_VEL
LIN {X 0,Y 767.779,Z 1065.314,A -85,B 0,C 180,E1 522.477,E2 522.477} C_VEL
LIN {X 0,Y 767.803,Z 1074.61,A -85,B 0,C 180,E1 523.088,E2 523.088} C_VEL
LIN {X 0,Y 767.75,Z 1084.792,A -85,B 0,C 180,E1 523.817,E2 523.817} C_VEL
LIN {X 0,Y 767.741,Z 1093.775,A -85,B 0,C 180,E1 524.519,E2 524.519} C_VEL
LIN {X 0,Y 767.824,Z 1101.772,A -85,B 0,C 180,E1 525.197,E2 525.197} C_VEL
LIN {X 0,Y 767.822,Z 1110.849,A -85,B 0,C 180,E1 526.037,E2 526.037} C_VEL
LIN {X 0,Y 767.788,Z 1118.688,A -85,B 0,C 180,E1 526.83,E2 526.83} C_VEL
LIN {X 0,Y 767.684,Z 1126.242,A -85,B 0,C 180,E1 527.665,E2 527.665} C_VEL
LIN {X 0,Y 767.739,Z 1133.09,A -85,B 0,C 180,E1 528.5,E2 528.5} C_VEL
LIN {X 0,Y 767.847,Z 1138.468,A -85,B 0,C 180,E1 529.214,E2 529.214} C_VEL
LIN {X 0,Y 767.649,Z 1144.953,A -85,B 0,C 180,E1 530.159,E2 530.159} C_VEL
LIN {X 0,Y 767.67,Z 1150.678,A -85,B 0,C 180,E1 531.105,E2 531.105} C_VEL
LIN {X 0,Y 767.82,Z 1155.701,A -85,B 0,C 180,E1 532.049,E2 532.049} C_VEL
LIN {X 0,Y 767.592,Z 1160.956,A -85,B 0,C 180,E1 533.188,E2 533.188} C_VEL
LIN {X 0,Y 767.6,Z 1161.315,A -85,B 0,C 180,E1 533.278,E2 533.278} C_VEL
LIN {X 0,Y 763.716,Z 1166.407,A -85,B 0,C 180,E1 534.508,E2 534.508} C_VEL
LIN {X 0,Y 759.772,Z 1170.193,A -85,B 0,C 180,E1 535.763,E2 535.763} C_VEL
LIN {X 0,Y 759.753,Z 1175.122,A -85,B 0,C 180,E1 538.859,E2 538.859} C_VEL
LIN {X 0,Y 759.763,Z 1175.045,A -85,B 0,C 180,E1 541.138,E2 541.138} C_VEL
LIN {X 0,Y 759.796,Z 1170.633,A -85,B 0,C 180,E1 543.99,E2 543.99} C_VEL
LIN {X 0,Y 759.882,Z 1159.817,A -85,B 0,C 180,E1 547.138,E2 547.138} C_VEL
LIN {X 0,Y 759.896,Z 1144.053,A -85,B 0,C 180,E1 550.019,E2 550.019} C_VEL
LIN {X 0,Y 759.952,Z 1123.015,A -85,B 0,C 180,E1 552.753,E2 552.753} C_VEL
LIN {X 0,Y 760.002,Z 1097.093,A -85,B 0,C 180,E1 555.273,E2 555.273} C_VEL
LIN {X 0,Y 760.101,Z 1066.649,A -85,B 0,C 180,E1 557.528,E2 557.528} C_VEL
LIN {X 0,Y 760.175,Z 1032.454,A -85,B 0,C 180,E1 559.447,E2 559.447} C_VEL
LIN {X 0,Y 760.291,Z 993.537,A -85,B 0,C 180,E1 561.037,E2 561.037} C_VEL
LIN {X 0,Y 760.392,Z 952.645,A -85,B 0,C 180,E1 562.144,E2 562.144} C_VEL
LIN {X 0,Y 759.468,Z 923.03,A -85,B 0,C 180,E1 562.673,E2 562.673} C_VEL
LIN {X 0,Y 759.715,Z 923.03,A -85,B 0,C 180,E1 568.512,E2 568.512} C_VEL
LIN {X 0,Y 759.582,Z 923.03,A -85,B 0,C 180,E1 573.354,E2 573.354} C_VEL
LIN {X 0,Y 759.382,Z 923.03,A -85,B 0,C 180,E1 578.086,E2 578.086} C_VEL
LIN {X 0,Y 759.711,Z 923.03,A -85,B 0,C 180,E1 582.633,E2 582.633} C_VEL
LIN {X 0,Y 759.666,Z 923.03,A -85,B 0,C 180,E1 587.462,E2 587.462} C_VEL
LIN {X 0,Y 759.688,Z 923.03,A -85,B 0,C 180,E1 593.38,E2 593.38} C_VEL
LIN {X 0,Y 759.614,Z 923.03,A -85,B 0,C 180,E1 597.528,E2 597.528} C_VEL
LIN {X 0,Y 759.712,Z 923.03,A -85,B 0,C 180,E1 601.501,E2 601.501} C_VEL
LIN {X 0,Y 759.819,Z 923.03,A -85,B 0,C 180,E1 606.682,E2 606.682} C_VEL
LIN {X 0,Y 760.402,Z 1001.759,A -85,B 0,C 180,E1 607.599,E2 607.599} C_VEL
LIN {X 0,Y 760.3,Z 1043.309,A -85,B 0,C 180,E1 608.593,E2 608.593} C_VEL
LIN {X 0,Y 760.197,Z 1080.512,A -85,B 0,C 180,E1 609.96,E2 609.96} C_VEL
LIN {X 0,Y 760.127,Z 1115.072,A -85,B 0,C 180,E1 611.714,E2 611.714} C_VEL
LIN {X 0,Y 760.073,Z 1146.811,A -85,B 0,C 180,E1 613.851,E2 613.851} C_VEL
LIN {X 0,Y 759.981,Z 1173.62,A -85,B 0,C 180,E1 616.208,E2 616.208} C_VEL
LIN {X 0,Y 759.919,Z 1196.312,A -85,B 0,C 180,E1 618.832,E2 618.832} C_VEL
LIN {X 0,Y 759.887,Z 1214.508,A -85,B 0,C 180,E1 621.722,E2 621.722} C_VEL
LIN {X 0,Y 759.841,Z 1225.69,A -85,B 0,C 180,E1 624.304,E2 624.304} C_VEL
LIN {X 0,Y 759.731,Z 1231.967,A -85,B 0,C 180,E1 626.59,E2 626.59} C_VEL
LIN {X 0,Y 759.76,Z 1235.092,A -85,B 0,C 180,E1 628.871,E2 628.871} C_VEL
LIN {X 0,Y 759.929,Z 1235.075,A -85,B 0,C 180,E1 631.149,E2 631.149} C_VEL
LIN {X 0,Y 759.798,Z 1230.721,A -85,B 0,C 180,E1 634.001,E2 634.001} C_VEL
LIN {X 0,Y 759.763,Z 1221.231,A -85,B 0,C 180,E1 636.863,E2 636.863} C_VEL
LIN {X 0,Y 759.798,Z 1206.145,A -85,B 0,C 180,E1 639.742,E2 639.742} C_VEL
LIN {X 0,Y 759.851,Z 1185.697,A -85,B 0,C 180,E1 642.499,E2 642.499} C_VEL
LIN {X 0,Y 759.942,Z 1159.253,A -85,B 0,C 180,E1 645.137,E2 645.137} C_VEL
LIN {X 0,Y 760.062,Z 1129.412,A -85,B 0,C 180,E1 647.393,E2 647.393} C_VEL
LIN {X 0,Y 760.203,Z 1096.182,A -85,B 0,C 180,E1 649.306,E2 649.306} C_VEL
LIN {X 0,Y 760.33,Z 1060.886,A -85,B 0,C 180,E1 650.818,E2 650.818} C_VEL
LIN {X 0,Y 760.401,Z 1024.293,A -85,B 0,C 180,E1 651.923,E2 651.923} C_VEL
LIN {X 0,Y 760.419,Z 984.848,A -85,B 0,C 180,E1 652.653,E2 652.653} C_VEL
LIN {X 0,Y 759.758,Z 923.03,A -85,B 0,C 180,E1 653.332,E2 653.332} C_VEL
LIN {X 0,Y 759.609,Z 923.03,A -85,B 0,C 180,E1 658.923,E2 658.923} C_VEL
LIN {X 0,Y 759.611,Z 923.03,A -85,B 0,C 180,E1 663.334,E2 663.334} C_VEL
LIN {X 0,Y 759.418,Z 923.03,A -85,B 0,C 180,E1 668.094,E2 668.094} C_VEL
LIN {X 0,Y 759.695,Z 923.03,A -85,B 0,C 180,E1 672.613,E2 672.613} C_VEL
LIN {X 0,Y 759.691,Z 923.03,A -85,B 0,C 180,E1 677.447,E2 677.447} C_VEL
LIN {X 0,Y 759.681,Z 923.03,A -85,B 0,C 180,E1 683.365,E2 683.365} C_VEL
LIN {X 0,Y 759.588,Z 923.03,A -85,B 0,C 180,E1 687.513,E2 687.513} C_VEL
LIN {X 0,Y 759.545,Z 923.03,A -85,B 0,C 180,E1 692.77,E2 692.77} C_VEL
LIN {X 0,Y 759.68,Z 923.03,A -85,B 0,C 180,E1 696.559,E2 696.559} C_VEL
LIN {X 0,Y 759.743,Z 923.03,A -85,B 0,C 180,E1 700.239,E2 700.239} C_VEL
LIN {X 0,Y 759.647,Z 923.03,A -85,B 0,C 180,E1 706.191,E2 706.191} C_VEL
LIN {X 0,Y 759.563,Z 923.03,A -85,B 0,C 180,E1 710.843,E2 710.843} C_VEL
LIN {X 0,Y 759.57,Z 923.03,A -85,B 0,C 180,E1 714.293,E2 714.293} C_VEL
LIN {X 0,Y 759.204,Z 923.03,A -85,B 0,C 180,E1 717.969,E2 717.969} C_VEL
LIN {X 0,Y 760.144,Z 969.387,A -85,B 0,C 180,E1 718.542,E2 718.542} C_VEL
LIN {X 0,Y 760.052,Z 998.155,A -85,B 0,C 180,E1 719.36,E2 719.36} C_VEL
LIN {X 0,Y 760.027,Z 1023.878,A -85,B 0,C 180,E1 720.571,E2 720.571} C_VEL
LIN {X 0,Y 759.994,Z 1046.164,A -85,B 0,C 180,E1 722.138,E2 722.138} C_VEL
LIN {X 0,Y 759.977,Z 1063.931,A -85,B 0,C 180,E1 723.992,E2 723.992} C_VEL
LIN {X 0,Y 759.945,Z 1076.932,A -85,B 0,C 180,E1 726.122,E2 726.122} C_VEL
LIN {X 0,Y 759.918,Z 1083.307,A -85,B 0,C 180,E1 728.002,E2 728.002} C_VEL
LIN {X 0,Y 759.929,Z 1085.403,A -85,B 0,C 180,E1 730.311,E2 730.311} C_VEL
LIN {X 0,Y 759.896,Z 1082.987,A -85,B 0,C 180,E1 732.053,E2 732.053} C_VEL
LIN {X 0,Y 759.895,Z 1075.471,A -85,B 0,C 180,E1 734.1,E2 734.1} C_VEL
LIN {X 0,Y 759.946,Z 1061.969,A -85,B 0,C 180,E1 736.165,E2 736.165} C_VEL
LIN {X 0,Y 759.977,Z 1043.915,A -85,B 0,C 180,E1 737.952,E2 737.952} C_VEL
LIN {X 0,Y 760.021,Z 1021.895,A -85,B 0,C 180,E1 739.454,E2 739.454} C_VEL
LIN {X 0,Y 760.063,Z 994.96,A -85,B 0,C 180,E1 740.666,E2 740.666} C_VEL
LIN {X 0,Y 760.121,Z 966.286,A -85,B 0,C 180,E1 741.427,E2 741.427} C_VEL
LIN {X 0,Y 759.356,Z 925.852,A -85,B 0,C 180,E1 741.901,E2 741.901} C_VEL
LIN {X 0,Y 759.121,Z 923.03,A -85,B 0,C 180,E1 741.993,E2 741.993} C_VEL
LIN {X 0,Y 759.703,Z 923.03,A -85,B 0,C 180,E1 745.952,E2 745.952} C_VEL
LIN {X 0,Y 759.565,Z 923.03,A -85,B 0,C 180,E1 751.18,E2 751.18} C_VEL
LIN {X 0,Y 759.584,Z 923.03,A -85,B 0,C 180,E1 755.339,E2 755.339} C_VEL
LIN {X 0,Y 759.807,Z 923.03,A -85,B 0,C 180,E1 759.526,E2 759.526} C_VEL
LIN {X 0,Y 759.621,Z 923.03,A -85,B 0,C 180,E1 765.865,E2 765.865} C_VEL
LIN {X 0,Y 759.698,Z 923.03,A -85,B 0,C 180,E1 770.874,E2 770.874} C_VEL
LIN {X 0,Y 759.445,Z 923.03,A -85,B 0,C 180,E1 776.134,E2 776.134} C_VEL
LIN {X 0,Y 759.456,Z 923.03,A -85,B 0,C 180,E1 781.103,E2 781.103} C_VEL
LIN {X 0,Y 759.834,Z 923.03,A -85,B 0,C 180,E1 784.046,E2 784.046} C_VEL
LIN {X 0,Y 759.528,Z 923.03,A -85,B 0,C 180,E1 789.007,E2 789.007} C_VEL
LIN {X 0,Y 759.552,Z 923.03,A -85,B 0,C 180,E1 793.819,E2 793.819} C_VEL
LIN {X 0,Y 759.467,Z 923.03,A -85,B 0,C 180,E1 798.514,E2 798.514} C_VEL
LIN {X 0,Y 759.548,Z 923.03,A -85,B 0,C 180,E1 801.985,E2 801.985} C_VEL
LIN {X 0,Y 759.762,Z 923.03,A -85,B 0,C 180,E1 806.57,E2 806.57} C_VEL
LIN {X 0,Y 759.886,Z 923.03,A -85,B 0,C 180,E1 811.129,E2 811.129} C_VEL
LIN {X 0,Y 759.575,Z 923.03,A -85,B 0,C 180,E1 815.89,E2 815.89} C_VEL
LIN {X 0,Y 759.533,Z 923.03,A -85,B 0,C 180,E1 820.304,E2 820.304} C_VEL
LIN {X 0,Y 759.504,Z 923.03,A -85,B 0,C 180,E1 823.801,E2 823.801} C_VEL
LIN {X 0,Y 759.604,Z 923.03,A -85,B 0,C 180,E1 827.349,E2 827.349} C_VEL
LIN {X 0,Y 759.514,Z 923.03,A -85,B 0,C 180,E1 830.972,E2 830.972} C_VEL
LIN {X 0,Y 759.598,Z 923.03,A -85,B 0,C 180,E1 834.68,E2 834.68} C_VEL
LIN {X 0,Y 759.587,Z 923.03,A -85,B 0,C 180,E1 838.915,E2 838.915} C_VEL
LIN {X 0,Y 759.614,Z 923.03,A -85,B 0,C 180,E1 843.329,E2 843.329} C_VEL
LIN {X 0,Y 759.405,Z 923.03,A -85,B 0,C 180,E1 848.07,E2 848.07} C_VEL
LIN {X 0,Y 759.792,Z 923.03,A -85,B 0,C 180,E1 852.618,E2 852.618} C_VEL
LIN {X 0,Y 759.595,Z 923.03,A -85,B 0,C 180,E1 855.87,E2 855.87} C_VEL
LIN {X 0,Y 759.689,Z 923.03,A -85,B 0,C 180,E1 860.851,E2 860.851} C_VEL
LIN {X 0,Y 759.45,Z 923.03,A -85,B 0,C 180,E1 866.141,E2 866.141} C_VEL
LIN {X 0,Y 759.446,Z 923.03,A -85,B 0,C 180,E1 871.072,E2 871.072} C_VEL
LIN {X 0,Y 759.855,Z 923.03,A -85,B 0,C 180,E1 874.054,E2 874.054} C_VEL
LIN {X 0,Y 759.832,Z 923.03,A -85,B 0,C 180,E1 877.258,E2 877.258} C_VEL
LIN {X 0,Y 760.422,Z 964.896,A -85,B 0,C 180,E1 878.046,E2 878.046} C_VEL
LIN {X 0,Y 760.277,Z 1002.348,A -85,B 0,C 180,E1 879.188,E2 879.188} C_VEL
LIN {X 0,Y 760.186,Z 1038.758,A -85,B 0,C 180,E1 880.777,E2 880.777} C_VEL
LIN {X 0,Y 760.105,Z 1073,A -85,B 0,C 180,E1 882.798,E2 882.798} C_VEL
LIN {X 0,Y 760.058,Z 1103.165,A -85,B 0,C 180,E1 885.168,E2 885.168} C_VEL
LIN {X 0,Y 759.86,Z 1127.344,A -85,B 0,C 180,E1 887.655,E2 887.655} C_VEL
LIN {X 0,Y 759.793,Z 1146.465,A -85,B 0,C 180,E1 890.266,E2 890.266} C_VEL
LIN {X 0,Y 759.78,Z 1160.224,A -85,B 0,C 180,E1 892.858,E2 892.858} C_VEL
LIN {X 0,Y 759.772,Z 1170.193,A -85,B 0,C 180,E1 895.763,E2 895.763} C_VEL
LIN {X 0,Y 755.779,Z 1172.97,A -85,B 0,C 180,E1 897.031,E2 897.031} C_VEL
LIN {X 0,Y 751.84,Z 1174.597,A -85,B 0,C 180,E1 898.324,E2 898.324} C_VEL
LIN {X 0,Y 751.863,Z 1175.046,A -85,B 0,C 180,E1 901.15,E2 901.15} C_VEL
LIN {X 0,Y 751.92,Z 1170.635,A -85,B 0,C 180,E1 904.032,E2 904.032} C_VEL
LIN {X 0,Y 752,Z 1159.821,A -85,B 0,C 180,E1 907.214,E2 907.214} C_VEL
LIN {X 0,Y 752.061,Z 1143.726,A -85,B 0,C 180,E1 910.174,E2 910.174} C_VEL
LIN {X 0,Y 752.113,Z 1122.063,A -85,B 0,C 180,E1 912.995,E2 912.995} C_VEL
LIN {X 0,Y 752.262,Z 1095.533,A -85,B 0,C 180,E1 915.568,E2 915.568} C_VEL
LIN {X 0,Y 752.455,Z 1064.851,A -85,B 0,C 180,E1 917.832,E2 917.832} C_VEL
LIN {X 0,Y 752.652,Z 1029.986,A -85,B 0,C 180,E1 919.773,E2 919.773} C_VEL
LIN {X 0,Y 752.882,Z 991.186,A -85,B 0,C 180,E1 921.331,E2 921.331} C_VEL
LIN {X 0,Y 753.066,Z 952.677,A -85,B 0,C 180,E1 922.371,E2 922.371} C_VEL
LIN {X 0,Y 751.957,Z 923.03,A -85,B 0,C 180,E1 922.913,E2 922.913} C_VEL
LIN {X 0,Y 751.733,Z 923.03,A -85,B 0,C 180,E1 928.843,E2 928.843} C_VEL
LIN {X 0,Y 751.803,Z 923.03,A -85,B 0,C 180,E1 932.865,E2 932.865} C_VEL
LIN {X 0,Y 751.752,Z 923.03,A -85,B 0,C 180,E1 937.086,E2 937.086} C_VEL
LIN {X 0,Y 751.622,Z 923.03,A -85,B 0,C 180,E1 943.12,E2 943.12} C_VEL
LIN {X 0,Y 751.496,Z 923.03,A -85,B 0,C 180,E1 948.446,E2 948.446} C_VEL
LIN {X 0,Y 751.747,Z 923.03,A -85,B 0,C 180,E1 953.516,E2 953.516} C_VEL
LIN {X 0,Y 751.474,Z 923.03,A -85,B 0,C 180,E1 958.494,E2 958.494} C_VEL
LIN {X 0,Y 751.547,Z 923.03,A -85,B 0,C 180,E1 962.469,E2 962.469} C_VEL
LIN {X 0,Y 751.795,Z 923.03,A -85,B 0,C 180,E1 966.411,E2 966.411} C_VEL
LIN {X 0,Y 753.046,Z 933.897,A -85,B 0,C 180,E1 966.577,E2 966.577} C_VEL
LIN {X 0,Y 753.101,Z 1001.439,A -85,B 0,C 180,E1 967.364,E2 967.364} C_VEL
LIN {X 0,Y 752.94,Z 1042.098,A -85,B 0,C 180,E1 968.334,E2 968.334} C_VEL
LIN {X 0,Y 752.694,Z 1080.169,A -85,B 0,C 180,E1 969.735,E2 969.735} C_VEL
LIN {X 0,Y 752.485,Z 1115.948,A -85,B 0,C 180,E1 971.574,E2 971.574} C_VEL
LIN {X 0,Y 752.352,Z 1146.811,A -85,B 0,C 180,E1 973.681,E2 973.681} C_VEL
LIN {X 0,Y 752.158,Z 1173.621,A -85,B 0,C 180,E1 976.061,E2 976.061} C_VEL
LIN {X 0,Y 752.046,Z 1196.313,A -85,B 0,C 180,E1 978.714,E2 978.714} C_VEL
LIN {X 0,Y 751.957,Z 1212.974,A -85,B 0,C 180,E1 981.343,E2 981.343} C_VEL
LIN {X 0,Y 751.943,Z 1225.69,A -85,B 0,C 180,E1 984.244,E2 984.244} C_VEL
LIN {X 0,Y 751.844,Z 1231.968,A -85,B 0,C 180,E1 986.554,E2 986.554} C_VEL
LIN {X 0,Y 751.861,Z 1235.093,A -85,B 0,C 180,E1 988.859,E2 988.859} C_VEL
LIN {X 0,Y 752.028,Z 1235.075,A -85,B 0,C 180,E1 991.161,E2 991.161} C_VEL
LIN {X 0,Y 751.925,Z 1230.721,A -85,B 0,C 180,E1 994.043,E2 994.043} C_VEL
LIN {X 0,Y 751.875,Z 1221.231,A -85,B 0,C 180,E1 996.936,E2 996.936} C_VEL
LIN {X 0,Y 751.953,Z 1205.74,A -85,B 0,C 180,E1 999.912,E2 999.912} C_VEL
LIN {X 0,Y 752.038,Z 1184.427,A -85,B 0,C 180,E1 1002.779,E2 1002.779} C_VEL
LIN {X 0,Y 752.224,Z 1158.355,A -85,B 0,C 180,E1 1005.373,E2 1005.373} C_VEL
LIN {X 0,Y 752.389,Z 1128.786,A -85,B 0,C 180,E1 1007.618,E2 1007.618} C_VEL
LIN {X 0,Y 752.651,Z 1094.805,A -85,B 0,C 180,E1 1009.577,E2 1009.577} C_VEL
LIN {X 0,Y 752.875,Z 1059.548,A -85,B 0,C 180,E1 1011.082,E2 1011.082} C_VEL
LIN {X 0,Y 753.084,Z 1022.664,A -85,B 0,C 180,E1 1012.186,E2 1012.186} C_VEL
LIN {X 0,Y 753.133,Z 984.72,A -85,B 0,C 180,E1 1012.887,E2 1012.887} C_VEL
LIN {X 0,Y 752.521,Z 926.326,A -85,B 0,C 180,E1 1013.518,E2 1013.518} C_VEL
LIN {X 0,Y 751.752,Z 923.03,A -85,B 0,C 180,E1 1013.636,E2 1013.636} C_VEL
LIN {X 0,Y 751.726,Z 923.03,A -85,B 0,C 180,E1 1018.854,E2 1018.854} C_VEL
LIN {X 0,Y 751.857,Z 923.03,A -85,B 0,C 180,E1 1022.873,E2 1022.873} C_VEL
LIN {X 0,Y 751.811,Z 923.03,A -85,B 0,C 180,E1 1027.092,E2 1027.092} C_VEL
LIN {X 0,Y 751.618,Z 923.03,A -85,B 0,C 180,E1 1033.131,E2 1033.131} C_VEL
LIN {X 0,Y 751.524,Z 923.03,A -85,B 0,C 180,E1 1038.432,E2 1038.432} C_VEL
LIN {X 0,Y 751.729,Z 923.03,A -85,B 0,C 180,E1 1043.53,E2 1043.53} C_VEL
LIN {X 0,Y 751.435,Z 923.03,A -85,B 0,C 180,E1 1048.478,E2 1048.478} C_VEL
LIN {X 0,Y 751.649,Z 923.03,A -85,B 0,C 180,E1 1052.46,E2 1052.46} C_VEL
LIN {X 0,Y 751.874,Z 923.03,A -85,B 0,C 180,E1 1056.301,E2 1056.301} C_VEL
LIN {X 0,Y 751.414,Z 923.03,A -85,B 0,C 180,E1 1061.232,E2 1061.232} C_VEL
LIN {X 0,Y 751.706,Z 923.03,A -85,B 0,C 180,E1 1066.042,E2 1066.042} C_VEL
LIN {X 0,Y 751.68,Z 923.03,A -85,B 0,C 180,E1 1070.747,E2 1070.747} C_VEL
LIN {X 0,Y 751.71,Z 923.03,A -85,B 0,C 180,E1 1074.233,E2 1074.233} C_VEL
LIN {X 0,Y 751.503,Z 923.03,A -85,B 0,C 180,E1 1077.841,E2 1077.841} C_VEL
LIN {X 0,Y 752.403,Z 969.158,A -85,B 0,C 180,E1 1078.419,E2 1078.419} C_VEL
LIN {X 0,Y 752.27,Z 997.086,A -85,B 0,C 180,E1 1079.21,E2 1079.21} C_VEL
LIN {X 0,Y 752.213,Z 1023.205,A -85,B 0,C 180,E1 1080.433,E2 1080.433} C_VEL
LIN {X 0,Y 752.127,Z 1045.698,A -85,B 0,C 180,E1 1082.016,E2 1082.016} C_VEL
LIN {X 0,Y 752.084,Z 1063.625,A -85,B 0,C 180,E1 1083.89,E2 1083.89} C_VEL
LIN {X 0,Y 752.003,Z 1075.467,A -85,B 0,C 180,E1 1085.768,E2 1085.768} C_VEL
LIN {X 0,Y 752.004,Z 1082.118,A -85,B 0,C 180,E1 1087.506,E2 1087.506} C_VEL
LIN {X 0,Y 751.995,Z 1085.481,A -85,B 0,C 180,E1 1090.03,E2 1090.03} C_VEL
LIN {X 0,Y 752.011,Z 1082.711,A -85,B 0,C 180,E1 1092.182,E2 1092.182} C_VEL
LIN {X 0,Y 752.017,Z 1074.921,A -85,B 0,C 180,E1 1094.251,E2 1094.251} C_VEL
LIN {X 0,Y 752.064,Z 1061.069,A -85,B 0,C 180,E1 1096.339,E2 1096.339} C_VEL
LIN {X 0,Y 752.112,Z 1042.544,A -85,B 0,C 180,E1 1098.146,E2 1098.146} C_VEL
LIN {X 0,Y 752.221,Z 1019.99,A -85,B 0,C 180,E1 1099.658,E2 1099.658} C_VEL
LIN {X 0,Y 752.279,Z 992.685,A -85,B 0,C 180,E1 1100.856,E2 1100.856} C_VEL
LIN {X 0,Y 752.378,Z 963.955,A -85,B 0,C 180,E1 1101.59,E2 1101.59} C_VEL
LIN {X 0,Y 751.387,Z 925.881,A -85,B 0,C 180,E1 1102.029,E2 1102.029} C_VEL
LIN {X 0,Y 751.291,Z 923.03,A -85,B 0,C 180,E1 1102.093,E2 1102.093} C_VEL
LIN {X 0,Y 751.737,Z 923.03,A -85,B 0,C 180,E1 1106.248,E2 1106.248} C_VEL
LIN {X 0,Y 751.586,Z 923.03,A -85,B 0,C 180,E1 1111.518,E2 1111.518} C_VEL
LIN {X 0,Y 751.454,Z 923.03,A -85,B 0,C 180,E1 1116.442,E2 1116.442} C_VEL
LIN {X 0,Y 751.659,Z 923.03,A -85,B 0,C 180,E1 1120.179,E2 1120.179} C_VEL
LIN {X 0,Y 751.689,Z 923.03,A -85,B 0,C 180,E1 1125.275,E2 1125.275} C_VEL
LIN {X 0,Y 751.741,Z 923.03,A -85,B 0,C 180,E1 1129.957,E2 1129.957} C_VEL
LIN {X 0,Y 751.536,Z 923.03,A -85,B 0,C 180,E1 1135.729,E2 1135.729} C_VEL
LIN {X 0,Y 751.672,Z 923.03,A -85,B 0,C 180,E1 1139.821,E2 1139.821} C_VEL
LIN {X 0,Y 751.674,Z 923.03,A -85,B 0,C 180,E1 1144.778,E2 1144.778} C_VEL
LIN {X 0,Y 751.648,Z 923.03,A -85,B 0,C 180,E1 1148.776,E2 1148.776} C_VEL
LIN {X 0,Y 751.649,Z 923.03,A -85,B 0,C 180,E1 1153.644,E2 1153.644} C_VEL
LIN {X 0,Y 751.542,Z 923.03,A -85,B 0,C 180,E1 1158.391,E2 1158.391} C_VEL
LIN {X 0,Y 751.882,Z 923.03,A -85,B 0,C 180,E1 1163.065,E2 1163.065} C_VEL
LIN {X 0,Y 751.888,Z 923.03,A -85,B 0,C 180,E1 1167.686,E2 1167.686} C_VEL
LIN {X 0,Y 751.707,Z 923.03,A -85,B 0,C 180,E1 1172.294,E2 1172.294} C_VEL
LIN {X 0,Y 751.717,Z 923.03,A -85,B 0,C 180,E1 1175.758,E2 1175.758} C_VEL
LIN {X 0,Y 751.64,Z 923.03,A -85,B 0,C 180,E1 1180.413,E2 1180.413} C_VEL
LIN {X 0,Y 751.594,Z 923.03,A -85,B 0,C 180,E1 1183.949,E2 1183.949} C_VEL
LIN {X 0,Y 751.667,Z 923.03,A -85,B 0,C 180,E1 1187.538,E2 1187.538} C_VEL
LIN {X 0,Y 751.564,Z 923.03,A -85,B 0,C 180,E1 1191.205,E2 1191.205} C_VEL
LIN {X 0,Y 751.601,Z 923.03,A -85,B 0,C 180,E1 1195.211,E2 1195.211} C_VEL
LIN {X 0,Y 751.707,Z 923.03,A -85,B 0,C 180,E1 1198.831,E2 1198.831} C_VEL
LIN {X 0,Y 751.831,Z 923.03,A -85,B 0,C 180,E1 1202.85,E2 1202.85} C_VEL
LIN {X 0,Y 751.76,Z 923.03,A -85,B 0,C 180,E1 1207.07,E2 1207.07} C_VEL
LIN {X 0,Y 751.827,Z 923.03,A -85,B 0,C 180,E1 1213.088,E2 1213.088} C_VEL
LIN {X 0,Y 751.433,Z 923.03,A -85,B 0,C 180,E1 1216.863,E2 1216.863} C_VEL
LIN {X 0,Y 751.566,Z 923.03,A -85,B 0,C 180,E1 1221.617,E2 1221.617} C_VEL
LIN {X 0,Y 751.542,Z 923.03,A -85,B 0,C 180,E1 1225.736,E2 1225.736} C_VEL
LIN {X 0,Y 751.679,Z 923.03,A -85,B 0,C 180,E1 1229.828,E2 1229.828} C_VEL
LIN {X 0,Y 751.724,Z 923.03,A -85,B 0,C 180,E1 1235.029,E2 1235.029} C_VEL
LIN {X 0,Y 751.895,Z 923.03,A -85,B 0,C 180,E1 1237.002,E2 1237.002} C_VEL
LIN {X 0,Y 753.073,Z 961.617,A -85,B 0,C 180,E1 1237.743,E2 1237.743} C_VEL
LIN {X 0,Y 752.837,Z 998.11,A -85,B 0,C 180,E1 1238.819,E2 1238.819} C_VEL
LIN {X 0,Y 752.668,Z 1033.586,A -85,B 0,C 180,E1 1240.317,E2 1240.317} C_VEL
LIN {X 0,Y 752.445,Z 1067.688,A -85,B 0,C 180,E1 1242.265,E2 1242.265} C_VEL
LIN {X 0,Y 752.228,Z 1098.259,A -85,B 0,C 180,E1 1244.573,E2 1244.573} C_VEL
LIN {X 0,Y 752.089,Z 1124.903,A -85,B 0,C 180,E1 1247.23,E2 1247.23} C_VEL
LIN {X 0,Y 751.967,Z 1145.476,A -85,B 0,C 180,E1 1250,E2 1250} C_VEL
LIN {X 0,Y 751.909,Z 1160.224,A -85,B 0,C 180,E1 1252.783,E2 1252.783} C_VEL
LIN {X 0,Y 751.884,Z 1170.294,A -85,B 0,C 180,E1 1255.757,E2 1255.757} C_VEL
LIN {X 0,Y 751.84,Z 1174.597,A -85,B 0,C 180,E1 1258.324,E2 1258.324} C_VEL
LIN {X 0,Y 749.273,Z 1175.359,A -85,B 0,C 180,E1 1259.306,E2 1259.306} C_VEL
LIN {X 0,Y 743.991,Z 1175.272,A -85,B 0,C 180,E1 1260.775,E2 1260.775} C_VEL
LIN {X 0,Y 743.923,Z 1175.131,A -85,B 0,C 180,E1 1260.944,E2 1260.944} C_VEL
LIN {X 0,Y 744.047,Z 1170.637,A -85,B 0,C 180,E1 1264.075,E2 1264.075} C_VEL
LIN {X 0,Y 744.12,Z 1159.824,A -85,B 0,C 180,E1 1267.29,E2 1267.29} C_VEL
LIN {X 0,Y 744.206,Z 1143.731,A -85,B 0,C 180,E1 1270.283,E2 1270.283} C_VEL
LIN {X 0,Y 744.309,Z 1122.935,A -85,B 0,C 180,E1 1273.036,E2 1273.036} C_VEL
LIN {X 0,Y 744.509,Z 1097.171,A -85,B 0,C 180,E1 1275.594,E2 1275.594} C_VEL
LIN {X 0,Y 744.782,Z 1067.143,A -85,B 0,C 180,E1 1277.87,E2 1277.87} C_VEL
LIN {X 0,Y 745.071,Z 1033.739,A -85,B 0,C 180,E1 1279.794,E2 1279.794} C_VEL
LIN {X 0,Y 745.385,Z 996.944,A -85,B 0,C 180,E1 1281.356,E2 1281.356} C_VEL
LIN {X 0,Y 745.715,Z 956.899,A -85,B 0,C 180,E1 1282.511,E2 1282.511} C_VEL
LIN {X 0,Y 744.605,Z 925.93,A -85,B 0,C 180,E1 1283.104,E2 1283.104} C_VEL
LIN {X 0,Y 744.011,Z 923.03,A -85,B 0,C 180,E1 1283.223,E2 1283.223} C_VEL
LIN {X 0,Y 743.744,Z 923.03,A -85,B 0,C 180,E1 1289.183,E2 1289.183} C_VEL
LIN {X 0,Y 743.714,Z 923.03,A -85,B 0,C 180,E1 1293.613,E2 1293.613} C_VEL
LIN {X 0,Y 743.675,Z 923.03,A -85,B 0,C 180,E1 1297.608,E2 1297.608} C_VEL
LIN {X 0,Y 743.717,Z 923.03,A -85,B 0,C 180,E1 1303.012,E2 1303.012} C_VEL
LIN {X 0,Y 743.697,Z 923.03,A -85,B 0,C 180,E1 1307.912,E2 1307.912} C_VEL
LIN {X 0,Y 743.755,Z 923.03,A -85,B 0,C 180,E1 1313.917,E2 1313.917} C_VEL
LIN {X 0,Y 743.571,Z 923.03,A -85,B 0,C 180,E1 1318.595,E2 1318.595} C_VEL
LIN {X 0,Y 743.749,Z 923.03,A -85,B 0,C 180,E1 1322.155,E2 1322.155} C_VEL
LIN {X 0,Y 743.773,Z 923.03,A -85,B 0,C 180,E1 1326.143,E2 1326.143} C_VEL
LIN {X 0,Y 745.831,Z 931.69,A -85,B 0,C 180,E1 1326.314,E2 1326.314} C_VEL
LIN {X 0,Y 745.784,Z 1000.067,A -85,B 0,C 180,E1 1327.107,E2 1327.107} C_VEL
LIN {X 0,Y 745.592,Z 1040.871,A -85,B 0,C 180,E1 1328.071,E2 1328.071} C_VEL
LIN {X 0,Y 745.195,Z 1080.338,A -85,B 0,C 180,E1 1329.53,E2 1329.53} C_VEL
LIN {X 0,Y 744.904,Z 1115.951,A -85,B 0,C 180,E1 1331.38,E2 1331.38} C_VEL
LIN {X 0,Y 744.626,Z 1146.811,A -85,B 0,C 180,E1 1333.507,E2 1333.507} C_VEL
LIN {X 0,Y 744.353,Z 1173.622,A -85,B 0,C 180,E1 1335.912,E2 1335.912} C_VEL
LIN {X 0,Y 744.21,Z 1196.314,A -85,B 0,C 180,E1 1338.593,E2 1338.593} C_VEL
LIN {X 0,Y 744.084,Z 1212.975,A -85,B 0,C 180,E1 1341.25,E2 1341.25} C_VEL
LIN {X 0,Y 744.044,Z 1225.691,A -85,B 0,C 180,E1 1344.183,E2 1344.183} C_VEL
LIN {X 0,Y 743.945,Z 1231.968,A -85,B 0,C 180,E1 1346.517,E2 1346.517} C_VEL
LIN {X 0,Y 743.962,Z 1235.093,A -85,B 0,C 180,E1 1348.847,E2 1348.847} C_VEL
LIN {X 0,Y 744.126,Z 1235.075,A -85,B 0,C 180,E1 1351.174,E2 1351.174} C_VEL
LIN {X 0,Y 744.05,Z 1230.721,A -85,B 0,C 180,E1 1354.086,E2 1354.086} C_VEL
LIN {X 0,Y 744.015,Z 1221.231,A -85,B 0,C 180,E1 1357.009,E2 1357.009} C_VEL
LIN {X 0,Y 744.085,Z 1206.14,A -85,B 0,C 180,E1 1359.951,E2 1359.951} C_VEL
LIN {X 0,Y 744.211,Z 1184.426,A -85,B 0,C 180,E1 1362.915,E2 1362.915} C_VEL
LIN {X 0,Y 744.47,Z 1158.355,A -85,B 0,C 180,E1 1365.537,E2 1365.537} C_VEL
LIN {X 0,Y 744.756,Z 1128.788,A -85,B 0,C 180,E1 1367.804,E2 1367.804} C_VEL
LIN {X 0,Y 745.103,Z 1094.986,A -85,B 0,C 180,E1 1369.774,E2 1369.774} C_VEL
LIN {X 0,Y 745.435,Z 1058.126,A -85,B 0,C 180,E1 1371.355,E2 1371.355} C_VEL
LIN {X 0,Y 745.765,Z 1021.035,A -85,B 0,C 180,E1 1372.455,E2 1372.455} C_VEL
LIN {X 0,Y 745.847,Z 982.806,A -85,B 0,C 180,E1 1373.146,E2 1373.146} C_VEL
LIN {X 0,Y 745.293,Z 928.115,A -85,B 0,C 180,E1 1373.741,E2 1373.741} C_VEL
LIN {X 0,Y 743.765,Z 923.03,A -85,B 0,C 180,E1 1373.902,E2 1373.902} C_VEL
LIN {X 0,Y 743.741,Z 923.03,A -85,B 0,C 180,E1 1379.193,E2 1379.193} C_VEL
LIN {X 0,Y 743.767,Z 923.03,A -85,B 0,C 180,E1 1383.595,E2 1383.595} C_VEL
LIN {X 0,Y 743.727,Z 923.03,A -85,B 0,C 180,E1 1387.592,E2 1387.592} C_VEL
LIN {X 0,Y 743.722,Z 923.03,A -85,B 0,C 180,E1 1392.994,E2 1392.994} C_VEL
LIN {X 0,Y 743.712,Z 923.03,A -85,B 0,C 180,E1 1397.896,E2 1397.896} C_VEL
LIN {X 0,Y 743.751,Z 923.03,A -85,B 0,C 180,E1 1403.901,E2 1403.901} C_VEL
LIN {X 0,Y 743.518,Z 923.03,A -85,B 0,C 180,E1 1408.615,E2 1408.615} C_VEL
LIN {X 0,Y 743.787,Z 923.03,A -85,B 0,C 180,E1 1412.144,E2 1412.144} C_VEL
LIN {X 0,Y 743.693,Z 923.03,A -85,B 0,C 180,E1 1417.292,E2 1417.292} C_VEL
LIN {X 0,Y 743.59,Z 923.03,A -85,B 0,C 180,E1 1421.027,E2 1421.027} C_VEL
LIN {X 0,Y 743.767,Z 923.03,A -85,B 0,C 180,E1 1425.89,E2 1425.89} C_VEL
LIN {X 0,Y 743.824,Z 923.03,A -85,B 0,C 180,E1 1430.648,E2 1430.648} C_VEL
LIN {X 0,Y 743.694,Z 923.03,A -85,B 0,C 180,E1 1434.689,E2 1434.689} C_VEL
LIN {X 0,Y 743.794,Z 923.03,A -85,B 0,C 180,E1 1437.709,E2 1437.709} C_VEL
LIN {X 0,Y 744.667,Z 968.923,A -85,B 0,C 180,E1 1438.293,E2 1438.293} C_VEL
LIN {X 0,Y 744.481,Z 997.93,A -85,B 0,C 180,E1 1439.129,E2 1439.129} C_VEL
LIN {X 0,Y 744.384,Z 1023.768,A -85,B 0,C 180,E1 1440.365,E2 1440.365} C_VEL
LIN {X 0,Y 744.294,Z 1045.215,A -85,B 0,C 180,E1 1441.892,E2 1441.892} C_VEL
LIN {X 0,Y 744.214,Z 1063.317,A -85,B 0,C 180,E1 1443.785,E2 1443.785} C_VEL
LIN {X 0,Y 744.13,Z 1075.947,A -85,B 0,C 180,E1 1445.829,E2 1445.829} C_VEL
LIN {X 0,Y 744.109,Z 1082.401,A -85,B 0,C 180,E1 1447.586,E2 1447.586} C_VEL
LIN {X 0,Y 744.096,Z 1085.287,A -85,B 0,C 180,E1 1449.351,E2 1449.351} C_VEL
LIN {X 0,Y 744.13,Z 1085.313,A -85,B 0,C 180,E1 1450.532,E2 1450.532} C_VEL
LIN {X 0,Y 744.132,Z 1080.66,A -85,B 0,C 180,E1 1452.909,E2 1452.909} C_VEL
LIN {X 0,Y 744.185,Z 1070.97,A -85,B 0,C 180,E1 1455.006,E2 1455.006} C_VEL
LIN {X 0,Y 744.272,Z 1055.322,A -85,B 0,C 180,E1 1457.057,E2 1457.057} C_VEL
LIN {X 0,Y 744.371,Z 1034.126,A -85,B 0,C 180,E1 1458.878,E2 1458.878} C_VEL
LIN {X 0,Y 744.442,Z 1009.659,A -85,B 0,C 180,E1 1460.286,E2 1460.286} C_VEL
LIN {X 0,Y 744.616,Z 981.245,A -85,B 0,C 180,E1 1461.324,E2 1461.324} C_VEL
LIN {X 0,Y 744.66,Z 952.643,A -85,B 0,C 180,E1 1461.876,E2 1461.876} C_VEL
LIN {X 0,Y 743.513,Z 923.03,A -85,B 0,C 180,E1 1462.19,E2 1462.19} C_VEL
LIN {X 0,Y 743.716,Z 923.03,A -85,B 0,C 180,E1 1466.607,E2 1466.607} C_VEL
LIN {X 0,Y 743.609,Z 923.03,A -85,B 0,C 180,E1 1471.895,E2 1471.895} C_VEL
LIN {X 0,Y 743.611,Z 923.03,A -85,B 0,C 180,E1 1476.11,E2 1476.11} C_VEL
LIN {X 0,Y 743.633,Z 923.03,A -85,B 0,C 180,E1 1480.562,E2 1480.562} C_VEL
LIN {X 0,Y 743.658,Z 923.03,A -85,B 0,C 180,E1 1486.292,E2 1486.292} C_VEL
LIN {X 0,Y 743.691,Z 923.03,A -85,B 0,C 180,E1 1490.949,E2 1490.949} C_VEL
LIN {X 0,Y 743.657,Z 923.03,A -85,B 0,C 180,E1 1495.314,E2 1495.314} C_VEL
LIN {X 0,Y 743.645,Z 923.03,A -85,B 0,C 180,E1 1500.803,E2 1500.803} C_VEL
LIN {X 0,Y 743.789,Z 923.03,A -85,B 0,C 180,E1 1504.737,E2 1504.737} C_VEL
LIN {X 0,Y 743.671,Z 923.03,A -85,B 0,C 180,E1 1509.182,E2 1509.182} C_VEL
LIN {X 0,Y 743.742,Z 923.03,A -85,B 0,C 180,E1 1513.465,E2 1513.465} C_VEL
LIN {X 0,Y 743.622,Z 923.03,A -85,B 0,C 180,E1 1518.266,E2 1518.266} C_VEL
LIN {X 0,Y 743.956,Z 923.03,A -85,B 0,C 180,E1 1522.99,E2 1522.99} C_VEL
LIN {X 0,Y 743.985,Z 923.03,A -85,B 0,C 180,E1 1527.662,E2 1527.662} C_VEL
LIN {X 0,Y 743.805,Z 923.03,A -85,B 0,C 180,E1 1532.318,E2 1532.318} C_VEL
LIN {X 0,Y 743.828,Z 923.03,A -85,B 0,C 180,E1 1535.819,E2 1535.819} C_VEL
LIN {X 0,Y 743.739,Z 923.03,A -85,B 0,C 180,E1 1540.525,E2 1540.525} C_VEL
LIN {X 0,Y 743.84,Z 923.03,A -85,B 0,C 180,E1 1545.301,E2 1545.301} C_VEL
LIN {X 0,Y 743.84,Z 923.03,A -85,B 0,C 180,E1 1550.19,E2 1550.19} C_VEL
LIN {X 0,Y 743.724,Z 923.03,A -85,B 0,C 180,E1 1555.243,E2 1555.243} C_VEL
LIN {X 0,Y 743.726,Z 923.03,A -85,B 0,C 180,E1 1559.17,E2 1559.17} C_VEL
LIN {X 0,Y 743.736,Z 923.03,A -85,B 0,C 180,E1 1563.587,E2 1563.587} C_VEL
LIN {X 0,Y 743.686,Z 923.03,A -85,B 0,C 180,E1 1567.584,E2 1567.584} C_VEL
LIN {X 0,Y 743.908,Z 923.03,A -85,B 0,C 180,E1 1573.005,E2 1573.005} C_VEL
LIN {X 0,Y 743.527,Z 923.03,A -85,B 0,C 180,E1 1577.003,E2 1577.003} C_VEL
LIN {X 0,Y 743.678,Z 923.03,A -85,B 0,C 180,E1 1580.956,E2 1580.956} C_VEL
LIN {X 0,Y 743.657,Z 923.03,A -85,B 0,C 180,E1 1585.321,E2 1585.321} C_VEL
LIN {X 0,Y 743.712,Z 923.03,A -85,B 0,C 180,E1 1589.471,E2 1589.471} C_VEL
LIN {X 0,Y 743.912,Z 923.03,A -85,B 0,C 180,E1 1594.749,E2 1594.749} C_VEL
LIN {X 0,Y 743.956,Z 923.03,A -85,B 0,C 180,E1 1596.748,E2 1596.748} C_VEL
LIN {X 0,Y 745.631,Z 934.066,A -85,B 0,C 180,E1 1596.96,E2 1596.96} C_VEL
LIN {X 0,Y 745.615,Z 973.67,A -85,B 0,C 180,E1 1597.822,E2 1597.822} C_VEL
LIN {X 0,Y 745.254,Z 1010.964,A -85,B 0,C 180,E1 1599.089,E2 1599.089} C_VEL
LIN {X 0,Y 744.96,Z 1046.952,A -85,B 0,C 180,E1 1600.813,E2 1600.813} C_VEL
LIN {X 0,Y 744.679,Z 1078.544,A -85,B 0,C 180,E1 1602.833,E2 1602.833} C_VEL
LIN {X 0,Y 744.452,Z 1107.972,A -85,B 0,C 180,E1 1605.301,E2 1605.301} C_VEL
LIN {X 0,Y 744.186,Z 1133.278,A -85,B 0,C 180,E1 1608.135,E2 1608.135} C_VEL
LIN {X 0,Y 744.045,Z 1151.61,A -85,B 0,C 180,E1 1610.943,E2 1610.943} C_VEL
LIN {X 0,Y 743.965,Z 1164.837,A -85,B 0,C 180,E1 1613.877,E2 1613.877} C_VEL
LIN {X 0,Y 743.951,Z 1172.038,A -85,B 0,C 180,E1 1616.505,E2 1616.505} C_VEL
LIN {X 0,Y 743.953,Z 1175.122,A -85,B 0,C 180,E1 1618.835,E2 1618.835} C_VEL
LIN {X 0,Y 743.923,Z 1175.131,A -85,B 0,C 180,E1 1620.944,E2 1620.944} C_VEL
LIN {X 0,Y 741.469,Z 1174.398,A -85,B 0,C 180,E1 1621.937,E2 1621.937} C_VEL
LIN {X 0,Y 736.153,Z 1172.108,A -85,B 0,C 180,E1 1623.409,E2 1623.409} C_VEL
LIN {X 0,Y 736.073,Z 1171.759,A -85,B 0,C 180,E1 1623.579,E2 1623.579} C_VEL
LIN {X 0,Y 736.15,Z 1163.391,A -85,B 0,C 180,E1 1626.481,E2 1626.481} C_VEL
LIN {X 0,Y 736.183,Z 1149.432,A -85,B 0,C 180,E1 1629.45,E2 1629.45} C_VEL
LIN {X 0,Y 736.395,Z 1130.262,A -85,B 0,C 180,E1 1632.291,E2 1632.291} C_VEL
LIN {X 0,Y 736.668,Z 1105.444,A -85,B 0,C 180,E1 1635.008,E2 1635.008} C_VEL
LIN {X 0,Y 736.958,Z 1076.811,A -85,B 0,C 180,E1 1637.39,E2 1637.39} C_VEL
LIN {X 0,Y 737.465,Z 1043.6,A -85,B 0,C 180,E1 1639.489,E2 1639.489} C_VEL
LIN {X 0,Y 737.903,Z 1006.5,A -85,B 0,C 180,E1 1641.224,E2 1641.224} C_VEL
LIN {X 0,Y 738.274,Z 966.16,A -85,B 0,C 180,E1 1642.527,E2 1642.527} C_VEL
LIN {X 0,Y 737.781,Z 929.077,A -85,B 0,C 180,E1 1643.289,E2 1643.289} C_VEL
LIN {X 0,Y 736.037,Z 923.03,A -85,B 0,C 180,E1 1643.465,E2 1643.465} C_VEL
LIN {X 0,Y 735.78,Z 923.03,A -85,B 0,C 180,E1 1649.53,E2 1649.53} C_VEL
LIN {X 0,Y 735.799,Z 923.03,A -85,B 0,C 180,E1 1653.674,E2 1653.674} C_VEL
LIN {X 0,Y 735.555,Z 923.03,A -85,B 0,C 180,E1 1658.702,E2 1658.702} C_VEL
LIN {X 0,Y 735.8,Z 923.03,A -85,B 0,C 180,E1 1662.663,E2 1662.663} C_VEL
LIN {X 0,Y 735.781,Z 923.03,A -85,B 0,C 180,E1 1667.674,E2 1667.674} C_VEL
LIN {X 0,Y 735.798,Z 923.03,A -85,B 0,C 180,E1 1673.464,E2 1673.464} C_VEL
LIN {X 0,Y 735.749,Z 923.03,A -85,B 0,C 180,E1 1677.74,E2 1677.74} C_VEL
LIN {X 0,Y 735.848,Z 923.03,A -85,B 0,C 180,E1 1682.007,E2 1682.007} C_VEL
LIN {X 0,Y 735.754,Z 923.03,A -85,B 0,C 180,E1 1685.861,E2 1685.861} C_VEL
LIN {X 0,Y 738.608,Z 933.915,A -85,B 0,C 180,E1 1686.091,E2 1686.091} C_VEL
LIN {X 0,Y 738.504,Z 1000.233,A -85,B 0,C 180,E1 1686.871,E2 1686.871} C_VEL
LIN {X 0,Y 738.237,Z 1040.871,A -85,B 0,C 180,E1 1687.841,E2 1687.841} C_VEL
LIN {X 0,Y 737.748,Z 1080.232,A -85,B 0,C 180,E1 1689.309,E2 1689.309} C_VEL
LIN {X 0,Y 737.33,Z 1115.953,A -85,B 0,C 180,E1 1691.181,E2 1691.181} C_VEL
LIN {X 0,Y 736.933,Z 1146.811,A -85,B 0,C 180,E1 1693.33,E2 1693.33} C_VEL
LIN {X 0,Y 736.553,Z 1173.623,A -85,B 0,C 180,E1 1695.76,E2 1695.76} C_VEL
LIN {X 0,Y 736.374,Z 1196.315,A -85,B 0,C 180,E1 1698.47,E2 1698.47} C_VEL
LIN {X 0,Y 736.189,Z 1212.975,A -85,B 0,C 180,E1 1701.156,E2 1701.156} C_VEL
LIN {X 0,Y 736.142,Z 1225.691,A -85,B 0,C 180,E1 1704.12,E2 1704.12} C_VEL
LIN {X 0,Y 736.048,Z 1231.968,A -85,B 0,C 180,E1 1706.48,E2 1706.48} C_VEL
LIN {X 0,Y 736.079,Z 1235.093,A -85,B 0,C 180,E1 1708.834,E2 1708.834} C_VEL
LIN {X 0,Y 736.231,Z 1235.076,A -85,B 0,C 180,E1 1711.186,E2 1711.186} C_VEL
LIN {X 0,Y 736.157,Z 1230.721,A -85,B 0,C 180,E1 1714.13,E2 1714.13} C_VEL
LIN {X 0,Y 736.127,Z 1221.231,A -85,B 0,C 180,E1 1717.085,E2 1717.085} C_VEL
LIN {X 0,Y 736.209,Z 1205.581,A -85,B 0,C 180,E1 1720.154,E2 1720.154} C_VEL
LIN {X 0,Y 736.421,Z 1184.424,A -85,B 0,C 180,E1 1723.054,E2 1723.054} C_VEL
LIN {X 0,Y 736.732,Z 1159.25,A -85,B 0,C 180,E1 1725.626,E2 1725.626} C_VEL
LIN {X 0,Y 737.094,Z 1128.79,A -85,B 0,C 180,E1 1727.996,E2 1727.996} C_VEL
LIN {X 0,Y 737.566,Z 1095.266,A -85,B 0,C 180,E1 1729.971,E2 1729.971} C_VEL
LIN {X 0,Y 737.99,Z 1059.877,A -85,B 0,C 180,E1 1731.517,E2 1731.517} C_VEL
LIN {X 0,Y 738.418,Z 1022.711,A -85,B 0,C 180,E1 1732.65,E2 1732.65} C_VEL
LIN {X 0,Y 738.589,Z 985.244,A -85,B 0,C 180,E1 1733.357,E2 1733.357} C_VEL
LIN {X 0,Y 738.174,Z 930.377,A -85,B 0,C 180,E1 1733.961,E2 1733.961} C_VEL
LIN {X 0,Y 735.753,Z 923.03,A -85,B 0,C 180,E1 1734.185,E2 1734.185} C_VEL
LIN {X 0,Y 735.777,Z 923.03,A -85,B 0,C 180,E1 1739.54,E2 1739.54} C_VEL
LIN {X 0,Y 735.847,Z 923.03,A -85,B 0,C 180,E1 1743.682,E2 1743.682} C_VEL
LIN {X 0,Y 735.544,Z 923.03,A -85,B 0,C 180,E1 1748.68,E2 1748.68} C_VEL
LIN {X 0,Y 735.82,Z 923.03,A -85,B 0,C 180,E1 1752.673,E2 1752.673} C_VEL
LIN {X 0,Y 735.822,Z 923.03,A -85,B 0,C 180,E1 1757.682,E2 1757.682} C_VEL
LIN {X 0,Y 735.798,Z 923.03,A -85,B 0,C 180,E1 1763.448,E2 1763.448} C_VEL
LIN {X 0,Y 735.703,Z 923.03,A -85,B 0,C 180,E1 1767.724,E2 1767.724} C_VEL
LIN {X 0,Y 735.867,Z 923.03,A -85,B 0,C 180,E1 1772.019,E2 1772.019} C_VEL
LIN {X 0,Y 735.818,Z 923.03,A -85,B 0,C 180,E1 1777.035,E2 1777.035} C_VEL
LIN {X 0,Y 735.727,Z 923.03,A -85,B 0,C 180,E1 1780.888,E2 1780.888} C_VEL
LIN {X 0,Y 735.829,Z 923.03,A -85,B 0,C 180,E1 1785.735,E2 1785.735} C_VEL
LIN {X 0,Y 735.928,Z 923.03,A -85,B 0,C 180,E1 1790.547,E2 1790.547} C_VEL
LIN {X 0,Y 735.932,Z 923.03,A -85,B 0,C 180,E1 1794.109,E2 1794.109} C_VEL
LIN {X 0,Y 735.977,Z 923.03,A -85,B 0,C 180,E1 1797.574,E2 1797.574} C_VEL
LIN {X 0,Y 736.923,Z 968.696,A -85,B 0,C 180,E1 1798.165,E2 1798.165} C_VEL
LIN {X 0,Y 736.74,Z 996.81,A -85,B 0,C 180,E1 1798.973,E2 1798.973} C_VEL
LIN {X 0,Y 736.579,Z 1023.094,A -85,B 0,C 180,E1 1800.222,E2 1800.222} C_VEL
LIN {X 0,Y 736.435,Z 1044.73,A -85,B 0,C 180,E1 1801.765,E2 1801.765} C_VEL
LIN {X 0,Y 736.345,Z 1063.01,A -85,B 0,C 180,E1 1803.678,E2 1803.678} C_VEL
LIN {X 0,Y 736.236,Z 1076.429,A -85,B 0,C 180,E1 1805.892,E2 1805.892} C_VEL
LIN {X 0,Y 736.227,Z 1082.677,A -85,B 0,C 180,E1 1807.668,E2 1807.668} C_VEL
LIN {X 0,Y 736.203,Z 1085.458,A -85,B 0,C 180,E1 1809.831,E2 1809.831} C_VEL
LIN {X 0,Y 736.233,Z 1082.297,A -85,B 0,C 180,E1 1812.389,E2 1812.389} C_VEL
LIN {X 0,Y 736.25,Z 1074.031,A -85,B 0,C 180,E1 1814.517,E2 1814.517} C_VEL
LIN {X 0,Y 736.345,Z 1060.52,A -85,B 0,C 180,E1 1816.544,E2 1816.544} C_VEL
LIN {X 0,Y 736.478,Z 1041.717,A -85,B 0,C 180,E1 1818.39,E2 1818.39} C_VEL
LIN {X 0,Y 736.596,Z 1018.228,A -85,B 0,C 180,E1 1819.961,E2 1819.961} C_VEL
LIN {X 0,Y 736.742,Z 991.898,A -85,B 0,C 180,E1 1821.117,E2 1821.117} C_VEL
LIN {X 0,Y 736.92,Z 963.291,A -85,B 0,C 180,E1 1821.85,E2 1821.85} C_VEL
LIN {X 0,Y 735.955,Z 926.361,A -85,B 0,C 180,E1 1822.282,E2 1822.282} C_VEL
LIN {X 0,Y 735.801,Z 923.03,A -85,B 0,C 180,E1 1822.387,E2 1822.387} C_VEL
LIN {X 0,Y 735.76,Z 923.03,A -85,B 0,C 180,E1 1826.863,E2 1826.863} C_VEL
LIN {X 0,Y 735.782,Z 923.03,A -85,B 0,C 180,E1 1830.894,E2 1830.894} C_VEL
LIN {X 0,Y 735.782,Z 923.03,A -85,B 0,C 180,E1 1835.104,E2 1835.104} C_VEL
LIN {X 0,Y 735.733,Z 923.03,A -85,B 0,C 180,E1 1840.532,E2 1840.532} C_VEL
LIN {X 0,Y 735.783,Z 923.03,A -85,B 0,C 180,E1 1845.958,E2 1845.958} C_VEL
LIN {X 0,Y 735.735,Z 923.03,A -85,B 0,C 180,E1 1851.305,E2 1851.305} C_VEL
LIN {X 0,Y 735.657,Z 923.03,A -85,B 0,C 180,E1 1856.308,E2 1856.308} C_VEL
LIN {X 0,Y 735.72,Z 923.03,A -85,B 0,C 180,E1 1860.457,E2 1860.457} C_VEL
LIN {X 0,Y 735.895,Z 923.03,A -85,B 0,C 180,E1 1864.625,E2 1864.625} C_VEL
LIN {X 0,Y 735.757,Z 923.03,A -85,B 0,C 180,E1 1869.556,E2 1869.556} C_VEL
LIN {X 0,Y 735.826,Z 923.03,A -85,B 0,C 180,E1 1874.507,E2 1874.507} C_VEL
LIN {X 0,Y 735.961,Z 923.03,A -85,B 0,C 180,E1 1880.255,E2 1880.255} C_VEL
LIN {X 0,Y 736.012,Z 923.03,A -85,B 0,C 180,E1 1884.098,E2 1884.098} C_VEL
LIN {X 0,Y 735.906,Z 923.03,A -85,B 0,C 180,E1 1888.813,E2 1888.813} C_VEL
LIN {X 0,Y 735.921,Z 923.03,A -85,B 0,C 180,E1 1892.343,E2 1892.343} C_VEL
LIN {X 0,Y 735.918,Z 923.03,A -85,B 0,C 180,E1 1895.882,E2 1895.882} C_VEL
LIN {X 0,Y 735.845,Z 923.03,A -85,B 0,C 180,E1 1900.639,E2 1900.639} C_VEL
LIN {X 0,Y 735.95,Z 923.03,A -85,B 0,C 180,E1 1905.469,E2 1905.469} C_VEL
LIN {X 0,Y 735.902,Z 923.03,A -85,B 0,C 180,E1 1910.418,E2 1910.418} C_VEL
LIN {X 0,Y 735.776,Z 923.03,A -85,B 0,C 180,E1 1915.535,E2 1915.535} C_VEL
LIN {X 0,Y 735.762,Z 923.03,A -85,B 0,C 180,E1 1919.517,E2 1919.517} C_VEL
LIN {X 0,Y 735.819,Z 923.03,A -85,B 0,C 180,E1 1923.659,E2 1923.659} C_VEL
LIN {X 0,Y 735.56,Z 923.03,A -85,B 0,C 180,E1 1928.678,E2 1928.678} C_VEL
LIN {X 0,Y 735.998,Z 923.03,A -85,B 0,C 180,E1 1934.06,E2 1934.06} C_VEL
LIN {X 0,Y 735.787,Z 923.03,A -85,B 0,C 180,E1 1939.431,E2 1939.431} C_VEL
LIN {X 0,Y 735.762,Z 923.03,A -85,B 0,C 180,E1 1944.895,E2 1944.895} C_VEL
LIN {X 0,Y 735.72,Z 923.03,A -85,B 0,C 180,E1 1950.465,E2 1950.465} C_VEL
LIN {X 0,Y 736.009,Z 923.03,A -85,B 0,C 180,E1 1954.568,E2 1954.568} C_VEL
LIN {X 0,Y 736.031,Z 923.03,A -85,B 0,C 180,E1 1956.48,E2 1956.48} C_VEL
LIN {X 0,Y 738.352,Z 934.319,A -85,B 0,C 180,E1 1956.725,E2 1956.725} C_VEL
LIN {X 0,Y 738.282,Z 973.659,A -85,B 0,C 180,E1 1957.59,E2 1957.59} C_VEL
LIN {X 0,Y 737.802,Z 1011.693,A -85,B 0,C 180,E1 1958.898,E2 1958.898} C_VEL
LIN {X 0,Y 737.369,Z 1047.839,A -85,B 0,C 180,E1 1960.658,E2 1960.658} C_VEL
LIN {X 0,Y 736.969,Z 1081.202,A -85,B 0,C 180,E1 1962.844,E2 1962.844} C_VEL
LIN {X 0,Y 736.651,Z 1111.009,A -85,B 0,C 180,E1 1965.445,E2 1965.445} C_VEL
LIN {X 0,Y 736.334,Z 1134.37,A -85,B 0,C 180,E1 1968.156,E2 1968.156} C_VEL
LIN {X 0,Y 736.162,Z 1151.605,A -85,B 0,C 180,E1 1970.845,E2 1970.845} C_VEL
LIN {X 0,Y 736.064,Z 1164.834,A -85,B 0,C 180,E1 1973.811,E2 1973.811} C_VEL
LIN {X 0,Y 736.053,Z 1172.038,A -85,B 0,C 180,E1 1976.468,E2 1976.468} C_VEL
LIN {X 0,Y 736.059,Z 1175.123,A -85,B 0,C 180,E1 1978.822,E2 1978.822} C_VEL
LIN {X 0,Y 736.068,Z 1175.048,A -85,B 0,C 180,E1 1981.175,E2 1981.175} C_VEL
LIN {X 0,Y 736.073,Z 1171.759,A -85,B 0,C 180,E1 1983.579,E2 1983.579} C_VEL
LIN {X 0,Y 734.859,Z 1170.332,A -85,B 0,C 180,E1 1984.244,E2 1984.244} C_VEL
LIN {X 0,Y 728.331,Z 1165.254,A -85,B 0,C 180,E1 1986.035,E2 1986.035} C_VEL
LIN {X 0,Y 728.251,Z 1164.699,A -85,B 0,C 180,E1 1986.203,E2 1986.203} C_VEL
LIN {X 0,Y 728.284,Z 1151.147,A -85,B 0,C 180,E1 1989.252,E2 1989.252} C_VEL
LIN {X 0,Y 728.558,Z 1131.866,A -85,B 0,C 180,E1 1992.224,E2 1992.224} C_VEL
LIN {X 0,Y 728.861,Z 1107.611,A -85,B 0,C 180,E1 1994.965,E2 1994.965} C_VEL
LIN {X 0,Y 729.248,Z 1079.079,A -85,B 0,C 180,E1 1997.411,E2 1997.411} C_VEL
LIN {X 0,Y 729.847,Z 1046.111,A -85,B 0,C 180,E1 1999.558,E2 1999.558} C_VEL
LIN {X 0,Y 730.429,Z 1009.986,A -85,B 0,C 180,E1 2001.307,E2 2001.307} C_VEL
LIN {X 0,Y 730.889,Z 972.078,A -85,B 0,C 180,E1 2002.604,E2 2002.604} C_VEL
LIN {X 0,Y 730.567,Z 931.095,A -85,B 0,C 180,E1 2003.501,E2 2003.501} C_VEL
LIN {X 0,Y 728.069,Z 923.03,A -85,B 0,C 180,E1 2003.748,E2 2003.748} C_VEL
LIN {X 0,Y 727.871,Z 923.03,A -85,B 0,C 180,E1 2009.346,E2 2009.346} C_VEL
LIN {X 0,Y 727.85,Z 923.03,A -85,B 0,C 180,E1 2014.092,E2 2014.092} C_VEL
LIN {X 0,Y 727.674,Z 923.03,A -85,B 0,C 180,E1 2018.533,E2 2018.533} C_VEL
LIN {X 0,Y 727.739,Z 923.03,A -85,B 0,C 180,E1 2023.406,E2 2023.406} C_VEL
LIN {X 0,Y 727.76,Z 923.03,A -85,B 0,C 180,E1 2028.38,E2 2028.38} C_VEL
LIN {X 0,Y 727.866,Z 923.03,A -85,B 0,C 180,E1 2034.061,E2 2034.061} C_VEL
LIN {X 0,Y 727.707,Z 923.03,A -85,B 0,C 180,E1 2038.742,E2 2038.742} C_VEL
LIN {X 0,Y 727.667,Z 923.03,A -85,B 0,C 180,E1 2043.244,E2 2043.244} C_VEL
LIN {X 0,Y 727.782,Z 923.03,A -85,B 0,C 180,E1 2045.581,E2 2045.581} C_VEL
LIN {X 0,Y 731.312,Z 933.336,A -85,B 0,C 180,E1 2045.831,E2 2045.831} C_VEL
LIN {X 0,Y 731.226,Z 1001.722,A -85,B 0,C 180,E1 2046.653,E2 2046.653} C_VEL
LIN {X 0,Y 730.831,Z 1042.278,A -85,B 0,C 180,E1 2047.65,E2 2047.65} C_VEL
LIN {X 0,Y 730.274,Z 1080.453,A -85,B 0,C 180,E1 2049.098,E2 2049.098} C_VEL
LIN {X 0,Y 729.682,Z 1115.955,A -85,B 0,C 180,E1 2050.977,E2 2050.977} C_VEL
LIN {X 0,Y 729.215,Z 1146.811,A -85,B 0,C 180,E1 2053.148,E2 2053.148} C_VEL
LIN {X 0,Y 728.766,Z 1173.624,A -85,B 0,C 180,E1 2055.604,E2 2055.604} C_VEL
LIN {X 0,Y 728.501,Z 1196.316,A -85,B 0,C 180,E1 2058.344,E2 2058.344} C_VEL
LIN {X 0,Y 728.344,Z 1214.509,A -85,B 0,C 180,E1 2061.36,E2 2061.36} C_VEL
LIN {X 0,Y 728.261,Z 1225.691,A -85,B 0,C 180,E1 2064.056,E2 2064.056} C_VEL
LIN {X 0,Y 728.152,Z 1231.969,A -85,B 0,C 180,E1 2066.441,E2 2066.441} C_VEL
LIN {X 0,Y 728.179,Z 1235.093,A -85,B 0,C 180,E1 2068.822,E2 2068.822} C_VEL
LIN {X 0,Y 728.33,Z 1235.076,A -85,B 0,C 180,E1 2071.199,E2 2071.199} C_VEL
LIN {X 0,Y 728.27,Z 1230.721,A -85,B 0,C 180,E1 2074.175,E2 2074.175} C_VEL
LIN {X 0,Y 728.305,Z 1219.976,A -85,B 0,C 180,E1 2077.461,E2 2077.461} C_VEL
LIN {X 0,Y 728.365,Z 1204.87,A -85,B 0,C 180,E1 2080.378,E2 2080.378} C_VEL
LIN {X 0,Y 728.66,Z 1183.1,A -85,B 0,C 180,E1 2083.348,E2 2083.348} C_VEL
LIN {X 0,Y 729.004,Z 1157.498,A -85,B 0,C 180,E1 2085.95,E2 2085.95} C_VEL
LIN {X 0,Y 729.488,Z 1127.653,A -85,B 0,C 180,E1 2088.268,E2 2088.268} C_VEL
LIN {X 0,Y 730.054,Z 1093.524,A -85,B 0,C 180,E1 2090.276,E2 2090.276} C_VEL
LIN {X 0,Y 730.64,Z 1056.656,A -85,B 0,C 180,E1 2091.865,E2 2091.865} C_VEL
LIN {X 0,Y 731.147,Z 1018.835,A -85,B 0,C 180,E1 2092.984,E2 2092.984} C_VEL
LIN {X 0,Y 731.39,Z 980.349,A -85,B 0,C 180,E1 2093.662,E2 2093.662} C_VEL
LIN {X 0,Y 730.942,Z 932.476,A -85,B 0,C 180,E1 2094.191,E2 2094.191} C_VEL
LIN {X 0,Y 727.805,Z 923.03,A -85,B 0,C 180,E1 2094.437,E2 2094.437} C_VEL
LIN {X 0,Y 727.867,Z 923.03,A -85,B 0,C 180,E1 2099.894,E2 2099.894} C_VEL
LIN {X 0,Y 727.876,Z 923.03,A -85,B 0,C 180,E1 2104.101,E2 2104.101} C_VEL
LIN {X 0,Y 727.67,Z 923.03,A -85,B 0,C 180,E1 2108.544,E2 2108.544} C_VEL
LIN {X 0,Y 727.768,Z 923.03,A -85,B 0,C 180,E1 2113.39,E2 2113.39} C_VEL
LIN {X 0,Y 727.768,Z 923.03,A -85,B 0,C 180,E1 2118.383,E2 2118.383} C_VEL
LIN {X 0,Y 727.862,Z 923.03,A -85,B 0,C 180,E1 2124.074,E2 2124.074} C_VEL
LIN {X 0,Y 727.68,Z 923.03,A -85,B 0,C 180,E1 2128.726,E2 2128.726} C_VEL
LIN {X 0,Y 727.823,Z 923.03,A -85,B 0,C 180,E1 2133.235,E2 2133.235} C_VEL
LIN {X 0,Y 727.912,Z 923.03,A -85,B 0,C 180,E1 2136.771,E2 2136.771} C_VEL
LIN {X 0,Y 727.838,Z 923.03,A -85,B 0,C 180,E1 2140.6,E2 2140.6} C_VEL
LIN {X 0,Y 727.917,Z 923.03,A -85,B 0,C 180,E1 2145.576,E2 2145.576} C_VEL
LIN {X 0,Y 728.045,Z 923.03,A -85,B 0,C 180,E1 2150.443,E2 2150.443} C_VEL
LIN {X 0,Y 727.841,Z 923.03,A -85,B 0,C 180,E1 2155.238,E2 2155.238} C_VEL
LIN {X 0,Y 728.043,Z 923.03,A -85,B 0,C 180,E1 2157.436,E2 2157.436} C_VEL
LIN {X 0,Y 729.212,Z 968.451,A -85,B 0,C 180,E1 2158.034,E2 2158.034} C_VEL
LIN {X 0,Y 728.952,Z 997.655,A -85,B 0,C 180,E1 2158.888,E2 2158.888} C_VEL
LIN {X 0,Y 728.751,Z 1023.658,A -85,B 0,C 180,E1 2160.15,E2 2160.15} C_VEL
LIN {X 0,Y 728.598,Z 1045.998,A -85,B 0,C 180,E1 2161.784,E2 2161.784} C_VEL
LIN {X 0,Y 728.473,Z 1063.785,A -85,B 0,C 180,E1 2163.718,E2 2163.718} C_VEL
LIN {X 0,Y 728.361,Z 1076.908,A -85,B 0,C 180,E1 2165.955,E2 2165.955} C_VEL
LIN {X 0,Y 728.337,Z 1082.904,A -85,B 0,C 180,E1 2167.752,E2 2167.752} C_VEL
LIN {X 0,Y 728.292,Z 1085.398,A -85,B 0,C 180,E1 2169.556,E2 2169.556} C_VEL
LIN {X 0,Y 728.331,Z 1083.312,A -85,B 0,C 180,E1 2171.976,E2 2171.976} C_VEL
LIN {X 0,Y 728.333,Z 1076.198,A -85,B 0,C 180,E1 2174.111,E2 2174.111} C_VEL
LIN {X 0,Y 728.424,Z 1063.25,A -85,B 0,C 180,E1 2176.265,E2 2176.265} C_VEL
LIN {X 0,Y 728.549,Z 1045.976,A -85,B 0,C 180,E1 2178.128,E2 2178.128} C_VEL
LIN {X 0,Y 728.775,Z 1023.482,A -85,B 0,C 180,E1 2179.771,E2 2179.771} C_VEL
LIN {X 0,Y 728.998,Z 997.7,A -85,B 0,C 180,E1 2181.02,E2 2181.02} C_VEL
LIN {X 0,Y 729.17,Z 968.573,A -85,B 0,C 180,E1 2181.873,E2 2181.873} C_VEL
LIN {X 0,Y 728.319,Z 927.753,A -85,B 0,C 180,E1 2182.399,E2 2182.399} C_VEL
LIN {X 0,Y 727.949,Z 923.03,A -85,B 0,C 180,E1 2182.466,E2 2182.466} C_VEL
LIN {X 0,Y 727.797,Z 923.03,A -85,B 0,C 180,E1 2187.181,E2 2187.181} C_VEL
LIN {X 0,Y 727.759,Z 923.03,A -85,B 0,C 180,E1 2191.634,E2 2191.634} C_VEL
LIN {X 0,Y 727.755,Z 923.03,A -85,B 0,C 180,E1 2195.914,E2 2195.914} C_VEL
LIN {X 0,Y 727.854,Z 923.03,A -85,B 0,C 180,E1 2200.062,E2 2200.062} C_VEL
LIN {X 0,Y 727.804,Z 923.03,A -85,B 0,C 180,E1 2205.086,E2 2205.086} C_VEL
LIN {X 0,Y 727.941,Z 923.03,A -85,B 0,C 180,E1 2210.182,E2 2210.182} C_VEL
LIN {X 0,Y 727.775,Z 923.03,A -85,B 0,C 180,E1 2216.155,E2 2216.155} C_VEL
LIN {X 0,Y 727.814,Z 923.03,A -85,B 0,C 180,E1 2221.467,E2 2221.467} C_VEL
LIN {X 0,Y 727.849,Z 923.03,A -85,B 0,C 180,E1 2225.995,E2 2225.995} C_VEL
LIN {X 0,Y 727.9,Z 923.03,A -85,B 0,C 180,E1 2230.591,E2 2230.591} C_VEL
LIN {X 0,Y 727.933,Z 923.03,A -85,B 0,C 180,E1 2235.566,E2 2235.566} C_VEL
LIN {X 0,Y 728.051,Z 923.03,A -85,B 0,C 180,E1 2240.432,E2 2240.432} C_VEL
LIN {X 0,Y 727.987,Z 923.03,A -85,B 0,C 180,E1 2245.227,E2 2245.227} C_VEL
LIN {X 0,Y 728.081,Z 923.03,A -85,B 0,C 180,E1 2249.99,E2 2249.99} C_VEL
LIN {X 0,Y 728.164,Z 923.03,A -85,B 0,C 180,E1 2255.046,E2 2255.046} C_VEL
LIN {X 0,Y 728.022,Z 923.03,A -85,B 0,C 180,E1 2259.547,E2 2259.547} C_VEL
LIN {X 0,Y 727.918,Z 923.03,A -85,B 0,C 180,E1 2264.413,E2 2264.413} C_VEL
LIN {X 0,Y 727.952,Z 923.03,A -85,B 0,C 180,E1 2268.129,E2 2268.129} C_VEL
LIN {X 0,Y 727.892,Z 923.03,A -85,B 0,C 180,E1 2273.217,E2 2273.217} C_VEL
LIN {X 0,Y 727.905,Z 923.03,A -85,B 0,C 180,E1 2278.505,E2 2278.505} C_VEL
LIN {X 0,Y 727.884,Z 923.03,A -85,B 0,C 180,E1 2283.857,E2 2283.857} C_VEL
LIN {X 0,Y 727.68,Z 923.03,A -85,B 0,C 180,E1 2288.516,E2 2288.516} C_VEL
LIN {X 0,Y 728.029,Z 923.03,A -85,B 0,C 180,E1 2293.408,E2 2293.408} C_VEL
LIN {X 0,Y 727.714,Z 923.03,A -85,B 0,C 180,E1 2298.356,E2 2298.356} C_VEL
LIN {X 0,Y 727.73,Z 923.03,A -85,B 0,C 180,E1 2302.973,E2 2302.973} C_VEL
LIN {X 0,Y 727.679,Z 923.03,A -85,B 0,C 180,E1 2307.321,E2 2307.321} C_VEL
LIN {X 0,Y 727.812,Z 923.03,A -85,B 0,C 180,E1 2311.474,E2 2311.474} C_VEL
LIN {X 0,Y 728.095,Z 923.03,A -85,B 0,C 180,E1 2316.211,E2 2316.211} C_VEL
LIN {X 0,Y 731.088,Z 934.856,A -85,B 0,C 180,E1 2316.489,E2 2316.489} C_VEL
LIN {X 0,Y 730.907,Z 975.251,A -85,B 0,C 180,E1 2317.398,E2 2317.398} C_VEL
LIN {X 0,Y 730.344,Z 1012.335,A -85,B 0,C 180,E1 2318.699,E2 2318.699} C_VEL
LIN {X 0,Y 729.778,Z 1047.836,A -85,B 0,C 180,E1 2320.449,E2 2320.449} C_VEL
LIN {X 0,Y 729.283,Z 1080.259,A -85,B 0,C 180,E1 2322.588,E2 2322.588} C_VEL
LIN {X 0,Y 728.878,Z 1109.892,A -85,B 0,C 180,E1 2325.172,E2 2325.172} C_VEL
LIN {X 0,Y 728.518,Z 1132.567,A -85,B 0,C 180,E1 2327.78,E2 2327.78} C_VEL
LIN {X 0,Y 728.273,Z 1151.6,A -85,B 0,C 180,E1 2330.745,E2 2330.745} C_VEL
LIN {X 0,Y 728.176,Z 1164.83,A -85,B 0,C 180,E1 2333.744,E2 2333.744} C_VEL
LIN {X 0,Y 728.155,Z 1172.039,A -85,B 0,C 180,E1 2336.429,E2 2336.429} C_VEL
LIN {X 0,Y 728.159,Z 1175.123,A -85,B 0,C 180,E1 2338.81,E2 2338.81} C_VEL
LIN {X 0,Y 728.168,Z 1175.049,A -85,B 0,C 180,E1 2341.188,E2 2341.188} C_VEL
LIN {X 0,Y 728.268,Z 1170.641,A -85,B 0,C 180,E1 2344.163,E2 2344.163} C_VEL
LIN {X 0,Y 728.251,Z 1164.699,A -85,B 0,C 180,E1 2346.203,E2 2346.203} C_VEL
LIN {X 0,Y 727.044,Z 1162.393,A -85,B 0,C 180,E1 2346.862,E2 2346.862} C_VEL
LIN {X 0,Y 720.506,Z 1154.884,A -85,B 0,C 180,E1 2348.618,E2 2348.618} C_VEL
LIN {X 0,Y 720.411,Z 1154.061,A -85,B 0,C 180,E1 2348.781,E2 2348.781} C_VEL
LIN {X 0,Y 720.617,Z 1137.016,A -85,B 0,C 180,E1 2351.643,E2 2351.643} C_VEL
LIN {X 0,Y 720.934,Z 1114.571,A -85,B 0,C 180,E1 2354.411,E2 2354.411} C_VEL
LIN {X 0,Y 721.472,Z 1088.062,A -85,B 0,C 180,E1 2356.893,E2 2356.893} C_VEL
LIN {X 0,Y 722.059,Z 1056.337,A -85,B 0,C 180,E1 2359.164,E2 2359.164} C_VEL
LIN {X 0,Y 722.812,Z 1022.282,A -85,B 0,C 180,E1 2360.998,E2 2360.998} C_VEL
LIN {X 0,Y 723.425,Z 985.536,A -85,B 0,C 180,E1 2362.438,E2 2362.438} C_VEL
LIN {X 0,Y 723.941,Z 947.275,A -85,B 0,C 180,E1 2363.438,E2 2363.438} C_VEL
LIN {X 0,Y 722.657,Z 931.242,A -85,B 0,C 180,E1 2363.772,E2 2363.772} C_VEL
LIN {X 0,Y 720.105,Z 923.03,A -85,B 0,C 180,E1 2363.994,E2 2363.994} C_VEL
LIN {X 0,Y 719.969,Z 923.03,A -85,B 0,C 180,E1 2368.863,E2 2368.863} C_VEL
LIN {X 0,Y 720.023,Z 923.03,A -85,B 0,C 180,E1 2373.068,E2 2373.068} C_VEL
LIN {X 0,Y 719.887,Z 923.03,A -85,B 0,C 180,E1 2377.496,E2 2377.496} C_VEL
LIN {X 0,Y 719.826,Z 923.03,A -85,B 0,C 180,E1 2382.736,E2 2382.736} C_VEL
LIN {X 0,Y 719.819,Z 923.03,A -85,B 0,C 180,E1 2387.816,E2 2387.816} C_VEL
LIN {X 0,Y 719.986,Z 923.03,A -85,B 0,C 180,E1 2392.894,E2 2392.894} C_VEL
LIN {X 0,Y 719.98,Z 923.03,A -85,B 0,C 180,E1 2397.087,E2 2397.087} C_VEL
LIN {X 0,Y 719.828,Z 923.03,A -85,B 0,C 180,E1 2402.509,E2 2402.509} C_VEL
LIN {X 0,Y 719.806,Z 923.03,A -85,B 0,C 180,E1 2405.29,E2 2405.29} C_VEL
LIN {X 0,Y 724.163,Z 936.731,A -85,B 0,C 180,E1 2405.613,E2 2405.613} C_VEL
LIN {X 0,Y 723.983,Z 1001.722,A -85,B 0,C 180,E1 2406.405,E2 2406.405} C_VEL
LIN {X 0,Y 723.468,Z 1043.042,A -85,B 0,C 180,E1 2407.436,E2 2407.436} C_VEL
LIN {X 0,Y 722.825,Z 1079.858,A -85,B 0,C 180,E1 2408.845,E2 2408.845} C_VEL
LIN {X 0,Y 722.13,Z 1114.691,A -85,B 0,C 180,E1 2410.691,E2 2410.691} C_VEL
LIN {X 0,Y 721.486,Z 1146.811,A -85,B 0,C 180,E1 2412.962,E2 2412.962} C_VEL
LIN {X 0,Y 720.953,Z 1173.625,A -85,B 0,C 180,E1 2415.445,E2 2415.445} C_VEL
LIN {X 0,Y 720.644,Z 1196.317,A -85,B 0,C 180,E1 2418.215,E2 2418.215} C_VEL
LIN {X 0,Y 720.456,Z 1214.51,A -85,B 0,C 180,E1 2421.265,E2 2421.265} C_VEL
LIN {X 0,Y 720.383,Z 1226.835,A -85,B 0,C 180,E1 2424.352,E2 2424.352} C_VEL
LIN {X 0,Y 720.278,Z 1231.969,A -85,B 0,C 180,E1 2426.402,E2 2426.402} C_VEL
LIN {X 0,Y 720.3,Z 1235.094,A -85,B 0,C 180,E1 2428.809,E2 2428.809} C_VEL
LIN {X 0,Y 720.44,Z 1235.076,A -85,B 0,C 180,E1 2431.212,E2 2431.212} C_VEL
LIN {X 0,Y 720.384,Z 1230.721,A -85,B 0,C 180,E1 2434.22,E2 2434.22} C_VEL
LIN {X 0,Y 720.452,Z 1219.976,A -85,B 0,C 180,E1 2437.543,E2 2437.543} C_VEL
LIN {X 0,Y 720.542,Z 1204.478,A -85,B 0,C 180,E1 2440.553,E2 2440.553} C_VEL
LIN {X 0,Y 720.843,Z 1183.098,A -85,B 0,C 180,E1 2443.496,E2 2443.496} C_VEL
LIN {X 0,Y 721.264,Z 1157.497,A -85,B 0,C 180,E1 2446.126,E2 2446.126} C_VEL
LIN {X 0,Y 721.863,Z 1127.655,A -85,B 0,C 180,E1 2448.468,E2 2448.468} C_VEL
LIN {X 0,Y 722.528,Z 1093.762,A -85,B 0,C 180,E1 2450.484,E2 2450.484} C_VEL
LIN {X 0,Y 723.247,Z 1056.652,A -85,B 0,C 180,E1 2452.1,E2 2452.1} C_VEL
LIN {X 0,Y 723.853,Z 1019.081,A -85,B 0,C 180,E1 2453.223,E2 2453.223} C_VEL
LIN {X 0,Y 724.156,Z 980.349,A -85,B 0,C 180,E1 2453.913,E2 2453.913} C_VEL
LIN {X 0,Y 723.669,Z 934.172,A -85,B 0,C 180,E1 2454.432,E2 2454.432} C_VEL
LIN {X 0,Y 719.842,Z 923.03,A -85,B 0,C 180,E1 2454.731,E2 2454.731} C_VEL
LIN {X 0,Y 719.956,Z 923.03,A -85,B 0,C 180,E1 2458.874,E2 2458.874} C_VEL
LIN {X 0,Y 720.042,Z 923.03,A -85,B 0,C 180,E1 2463.078,E2 2463.078} C_VEL
LIN {X 0,Y 719.916,Z 923.03,A -85,B 0,C 180,E1 2467.505,E2 2467.505} C_VEL
LIN {X 0,Y 719.826,Z 923.03,A -85,B 0,C 180,E1 2472.717,E2 2472.717} C_VEL
LIN {X 0,Y 719.818,Z 923.03,A -85,B 0,C 180,E1 2477.798,E2 2477.798} C_VEL
LIN {X 0,Y 719.984,Z 923.03,A -85,B 0,C 180,E1 2482.906,E2 2482.906} C_VEL
LIN {X 0,Y 719.937,Z 923.03,A -85,B 0,C 180,E1 2487.106,E2 2487.106} C_VEL
LIN {X 0,Y 719.917,Z 923.03,A -85,B 0,C 180,E1 2492.5,E2 2492.5} C_VEL
LIN {X 0,Y 719.935,Z 923.03,A -85,B 0,C 180,E1 2497.463,E2 2497.463} C_VEL
LIN {X 0,Y 719.702,Z 923.03,A -85,B 0,C 180,E1 2501.644,E2 2501.644} C_VEL
LIN {X 0,Y 719.938,Z 923.03,A -85,B 0,C 180,E1 2506.652,E2 2506.652} C_VEL
LIN {X 0,Y 720.132,Z 923.03,A -85,B 0,C 180,E1 2510.513,E2 2510.513} C_VEL
LIN {X 0,Y 719.944,Z 923.03,A -85,B 0,C 180,E1 2515.185,E2 2515.185} C_VEL
LIN {X 0,Y 720.149,Z 923.03,A -85,B 0,C 180,E1 2517.316,E2 2517.316} C_VEL
LIN {X 0,Y 721.506,Z 960.251,A -85,B 0,C 180,E1 2517.751,E2 2517.751} C_VEL
LIN {X 0,Y 721.277,Z 990.528,A -85,B 0,C 180,E1 2518.501,E2 2518.501} C_VEL
LIN {X 0,Y 720.997,Z 1017.686,A -85,B 0,C 180,E1 2519.701,E2 2519.701} C_VEL
LIN {X 0,Y 720.787,Z 1040.087,A -85,B 0,C 180,E1 2521.203,E2 2521.203} C_VEL
LIN {X 0,Y 720.602,Z 1058.674,A -85,B 0,C 180,E1 2523.006,E2 2523.006} C_VEL
LIN {X 0,Y 720.498,Z 1072.637,A -85,B 0,C 180,E1 2525.033,E2 2525.033} C_VEL
LIN {X 0,Y 720.448,Z 1081.678,A -85,B 0,C 180,E1 2527.231,E2 2527.231} C_VEL
LIN {X 0,Y 720.407,Z 1085.429,A -85,B 0,C 180,E1 2529.662,E2 2529.662} C_VEL
LIN {X 0,Y 720.431,Z 1083.051,A -85,B 0,C 180,E1 2532.109,E2 2532.109} C_VEL
LIN {X 0,Y 720.451,Z 1075.674,A -85,B 0,C 180,E1 2534.269,E2 2534.269} C_VEL
LIN {X 0,Y 720.576,Z 1062.424,A -85,B 0,C 180,E1 2536.447,E2 2536.447} C_VEL
LIN {X 0,Y 720.727,Z 1044.677,A -85,B 0,C 180,E1 2538.332,E2 2538.332} C_VEL
LIN {X 0,Y 720.958,Z 1022.849,A -85,B 0,C 180,E1 2539.914,E2 2539.914} C_VEL
LIN {X 0,Y 721.209,Z 995.884,A -85,B 0,C 180,E1 2541.209,E2 2541.209} C_VEL
LIN {X 0,Y 721.455,Z 967.584,A -85,B 0,C 180,E1 2542.023,E2 2542.023} C_VEL
LIN {X 0,Y 720.573,Z 927.874,A -85,B 0,C 180,E1 2542.534,E2 2542.534} C_VEL
LIN {X 0,Y 720.072,Z 923.03,A -85,B 0,C 180,E1 2542.626,E2 2542.626} C_VEL
LIN {X 0,Y 719.834,Z 923.03,A -85,B 0,C 180,E1 2547.507,E2 2547.507} C_VEL
LIN {X 0,Y 719.857,Z 923.03,A -85,B 0,C 180,E1 2551.656,E2 2551.656} C_VEL
LIN {X 0,Y 719.842,Z 923.03,A -85,B 0,C 180,E1 2556.001,E2 2556.001} C_VEL
LIN {X 0,Y 719.746,Z 923.03,A -85,B 0,C 180,E1 2560.893,E2 2560.893} C_VEL
LIN {X 0,Y 719.804,Z 923.03,A -85,B 0,C 180,E1 2566.14,E2 2566.14} C_VEL
LIN {X 0,Y 719.916,Z 923.03,A -85,B 0,C 180,E1 2570.963,E2 2570.963} C_VEL
LIN {X 0,Y 719.832,Z 923.03,A -85,B 0,C 180,E1 2575.464,E2 2575.464} C_VEL
LIN {X 0,Y 719.889,Z 923.03,A -85,B 0,C 180,E1 2579.741,E2 2579.741} C_VEL
LIN {X 0,Y 720.033,Z 923.03,A -85,B 0,C 180,E1 2584.481,E2 2584.481} C_VEL
LIN {X 0,Y 719.978,Z 923.03,A -85,B 0,C 180,E1 2589.087,E2 2589.087} C_VEL
LIN {X 0,Y 720.001,Z 923.03,A -85,B 0,C 180,E1 2594.157,E2 2594.157} C_VEL
LIN {X 0,Y 720.177,Z 923.03,A -85,B 0,C 180,E1 2599.105,E2 2599.105} C_VEL
LIN {X 0,Y 720.205,Z 923.03,A -85,B 0,C 180,E1 2603.968,E2 2603.968} C_VEL
LIN {X 0,Y 720.139,Z 923.03,A -85,B 0,C 180,E1 2608.787,E2 2608.787} C_VEL
LIN {X 0,Y 720.116,Z 923.03,A -85,B 0,C 180,E1 2612.394,E2 2612.394} C_VEL
LIN {X 0,Y 720.118,Z 923.03,A -85,B 0,C 180,E1 2616.011,E2 2616.011} C_VEL
LIN {X 0,Y 720.056,Z 923.03,A -85,B 0,C 180,E1 2620.875,E2 2620.875} C_VEL
LIN {X 0,Y 720.144,Z 923.03,A -85,B 0,C 180,E1 2625.817,E2 2625.817} C_VEL
LIN {X 0,Y 720.017,Z 923.03,A -85,B 0,C 180,E1 2630.889,E2 2630.889} C_VEL
LIN {X 0,Y 719.962,Z 923.03,A -85,B 0,C 180,E1 2636.138,E2 2636.138} C_VEL
LIN {X 0,Y 719.893,Z 923.03,A -85,B 0,C 180,E1 2640.612,E2 2640.612} C_VEL
LIN {X 0,Y 719.82,Z 923.03,A -85,B 0,C 180,E1 2645.041,E2 2645.041} C_VEL
LIN {X 0,Y 719.748,Z 923.03,A -85,B 0,C 180,E1 2649.029,E2 2649.029} C_VEL
LIN {X 0,Y 720.098,Z 923.03,A -85,B 0,C 180,E1 2653.808,E2 2653.808} C_VEL
LIN {X 0,Y 719.86,Z 923.03,A -85,B 0,C 180,E1 2659.401,E2 2659.401} C_VEL
LIN {X 0,Y 719.851,Z 923.03,A -85,B 0,C 180,E1 2663.999,E2 2663.999} C_VEL
LIN {X 0,Y 719.87,Z 923.03,A -85,B 0,C 180,E1 2669.359,E2 2669.359} C_VEL
LIN {X 0,Y 720.122,Z 923.03,A -85,B 0,C 180,E1 2674.427,E2 2674.427} C_VEL
LIN {X 0,Y 720.17,Z 923.03,A -85,B 0,C 180,E1 2675.931,E2 2675.931} C_VEL
LIN {X 0,Y 723.867,Z 937.189,A -85,B 0,C 180,E1 2676.279,E2 2676.279} C_VEL
LIN {X 0,Y 723.505,Z 977.788,A -85,B 0,C 180,E1 2677.228,E2 2677.228} C_VEL
LIN {X 0,Y 722.853,Z 1016.51,A -85,B 0,C 180,E1 2678.647,E2 2678.647} C_VEL
LIN {X 0,Y 722.098,Z 1052.628,A -85,B 0,C 180,E1 2680.516,E2 2680.516} C_VEL
LIN {X 0,Y 721.512,Z 1085.087,A -85,B 0,C 180,E1 2682.774,E2 2682.774} C_VEL
LIN {X 0,Y 721.062,Z 1112.805,A -85,B 0,C 180,E1 2685.314,E2 2685.314} C_VEL
LIN {X 0,Y 720.642,Z 1135.457,A -85,B 0,C 180,E1 2688.048,E2 2688.048} C_VEL
LIN {X 0,Y 720.422,Z 1153.146,A -85,B 0,C 180,E1 2690.948,E2 2690.948} C_VEL
LIN {X 0,Y 720.306,Z 1165.802,A -85,B 0,C 180,E1 2693.978,E2 2693.978} C_VEL
LIN {X 0,Y 720.272,Z 1172.039,A -85,B 0,C 180,E1 2696.39,E2 2696.39} C_VEL
LIN {X 0,Y 720.27,Z 1175.123,A -85,B 0,C 180,E1 2698.797,E2 2698.797} C_VEL
LIN {X 0,Y 720.279,Z 1175.049,A -85,B 0,C 180,E1 2701.201,E2 2701.201} C_VEL
LIN {X 0,Y 720.401,Z 1170.642,A -85,B 0,C 180,E1 2704.209,E2 2704.209} C_VEL
LIN {X 0,Y 720.517,Z 1159.836,A -85,B 0,C 180,E1 2707.531,E2 2707.531} C_VEL
LIN {X 0,Y 720.411,Z 1154.061,A -85,B 0,C 180,E1 2708.781,E2 2708.781} C_VEL
LIN {X 0,Y 716.588,Z 1147.56,A -85,B 0,C 180,E1 2710.043,E2 2710.043} C_VEL
LIN {X 0,Y 712.762,Z 1140.262,A -85,B 0,C 180,E1 2711.291,E2 2711.291} C_VEL
LIN {X 0,Y 713.104,Z 1117.452,A -85,B 0,C 180,E1 2714.26,E2 2714.26} C_VEL
LIN {X 0,Y 713.724,Z 1089.984,A -85,B 0,C 180,E1 2716.923,E2 2716.923} C_VEL
LIN {X 0,Y 714.448,Z 1057.6,A -85,B 0,C 180,E1 2719.296,E2 2719.296} C_VEL
LIN {X 0,Y 715.339,Z 1022.539,A -85,B 0,C 180,E1 2721.216,E2 2721.216} C_VEL
LIN {X 0,Y 716.079,Z 985.095,A -85,B 0,C 180,E1 2722.696,E2 2722.696} C_VEL
LIN {X 0,Y 716.662,Z 946.918,A -85,B 0,C 180,E1 2723.698,E2 2723.698} C_VEL
LIN {X 0,Y 715.512,Z 933.456,A -85,B 0,C 180,E1 2723.987,E2 2723.987} C_VEL
LIN {X 0,Y 712.114,Z 923.03,A -85,B 0,C 180,E1 2724.315,E2 2724.315} C_VEL
LIN {X 0,Y 711.995,Z 923.03,A -85,B 0,C 180,E1 2729.554,E2 2729.554} C_VEL
LIN {X 0,Y 711.988,Z 923.03,A -85,B 0,C 180,E1 2734.162,E2 2734.162} C_VEL
LIN {X 0,Y 711.863,Z 923.03,A -85,B 0,C 180,E1 2738.265,E2 2738.265} C_VEL
LIN {X 0,Y 711.933,Z 923.03,A -85,B 0,C 180,E1 2742.78,E2 2742.78} C_VEL
LIN {X 0,Y 711.907,Z 923.03,A -85,B 0,C 180,E1 2747.978,E2 2747.978} C_VEL
LIN {X 0,Y 712.065,Z 923.03,A -85,B 0,C 180,E1 2753.744,E2 2753.744} C_VEL
LIN {X 0,Y 711.961,Z 923.03,A -85,B 0,C 180,E1 2758.098,E2 2758.098} C_VEL
LIN {X 0,Y 711.838,Z 923.03,A -85,B 0,C 180,E1 2763.07,E2 2763.07} C_VEL
LIN {X 0,Y 711.857,Z 923.03,A -85,B 0,C 180,E1 2765.002,E2 2765.002} C_VEL
LIN {X 0,Y 716.934,Z 937.368,A -85,B 0,C 180,E1 2765.358,E2 2765.358} C_VEL
LIN {X 0,Y 716.738,Z 1001.198,A -85,B 0,C 180,E1 2766.142,E2 2766.142} C_VEL
LIN {X 0,Y 716.176,Z 1042.281,A -85,B 0,C 180,E1 2767.168,E2 2767.168} C_VEL
LIN {X 0,Y 715.361,Z 1080.317,A -85,B 0,C 180,E1 2768.635,E2 2768.635} C_VEL
LIN {X 0,Y 714.58,Z 1114.687,A -85,B 0,C 180,E1 2770.478,E2 2770.478} C_VEL
LIN {X 0,Y 713.793,Z 1146.811,A -85,B 0,C 180,E1 2772.773,E2 2772.773} C_VEL
LIN {X 0,Y 713.187,Z 1173.626,A -85,B 0,C 180,E1 2775.283,E2 2775.283} C_VEL
LIN {X 0,Y 712.821,Z 1196.318,A -85,B 0,C 180,E1 2778.084,E2 2778.084} C_VEL
LIN {X 0,Y 712.581,Z 1214.648,A -85,B 0,C 180,E1 2781.196,E2 2781.196} C_VEL
LIN {X 0,Y 712.475,Z 1225.691,A -85,B 0,C 180,E1 2783.924,E2 2783.924} C_VEL
LIN {X 0,Y 712.382,Z 1231.969,A -85,B 0,C 180,E1 2786.363,E2 2786.363} C_VEL
LIN {X 0,Y 712.4,Z 1235.094,A -85,B 0,C 180,E1 2788.795,E2 2788.795} C_VEL
LIN {X 0,Y 712.538,Z 1235.077,A -85,B 0,C 180,E1 2791.226,E2 2791.226} C_VEL
LIN {X 0,Y 712.479,Z 1229.924,A -85,B 0,C 180,E1 2794.584,E2 2794.584} C_VEL
LIN {X 0,Y 712.572,Z 1219.976,A -85,B 0,C 180,E1 2797.626,E2 2797.626} C_VEL
LIN {X 0,Y 712.694,Z 1204.283,A -85,B 0,C 180,E1 2800.701,E2 2800.701} C_VEL
LIN {X 0,Y 713.058,Z 1183.097,A -85,B 0,C 180,E1 2803.646,E2 2803.646} C_VEL
LIN {X 0,Y 713.532,Z 1157.496,A -85,B 0,C 180,E1 2806.306,E2 2806.306} C_VEL
LIN {X 0,Y 714.272,Z 1127.677,A -85,B 0,C 180,E1 2808.67,E2 2808.67} C_VEL
LIN {X 0,Y 715.023,Z 1094.678,A -85,B 0,C 180,E1 2810.66,E2 2810.66} C_VEL
LIN {X 0,Y 715.845,Z 1058.121,A -85,B 0,C 180,E1 2812.285,E2 2812.285} C_VEL
LIN {X 0,Y 716.545,Z 1020.537,A -85,B 0,C 180,E1 2813.437,E2 2813.437} C_VEL
LIN {X 0,Y 716.939,Z 981.655,A -85,B 0,C 180,E1 2814.152,E2 2814.152} C_VEL
LIN {X 0,Y 716.554,Z 936.432,A -85,B 0,C 180,E1 2814.666,E2 2814.666} C_VEL
LIN {X 0,Y 711.883,Z 923.03,A -85,B 0,C 180,E1 2815.049,E2 2815.049} C_VEL
LIN {X 0,Y 711.991,Z 923.03,A -85,B 0,C 180,E1 2819.525,E2 2819.525} C_VEL
LIN {X 0,Y 711.995,Z 923.03,A -85,B 0,C 180,E1 2824.138,E2 2824.138} C_VEL
LIN {X 0,Y 711.853,Z 923.03,A -85,B 0,C 180,E1 2828.242,E2 2828.242} C_VEL
LIN {X 0,Y 711.94,Z 923.03,A -85,B 0,C 180,E1 2832.791,E2 2832.791} C_VEL
LIN {X 0,Y 711.908,Z 923.03,A -85,B 0,C 180,E1 2837.99,E2 2837.99} C_VEL
LIN {X 0,Y 712.067,Z 923.03,A -85,B 0,C 180,E1 2843.757,E2 2843.757} C_VEL
LIN {X 0,Y 711.912,Z 923.03,A -85,B 0,C 180,E1 2848.119,E2 2848.119} C_VEL
LIN {X 0,Y 711.981,Z 923.03,A -85,B 0,C 180,E1 2853.063,E2 2853.063} C_VEL
LIN {X 0,Y 712.053,Z 923.03,A -85,B 0,C 180,E1 2857.544,E2 2857.544} C_VEL
LIN {X 0,Y 711.842,Z 923.03,A -85,B 0,C 180,E1 2861.434,E2 2861.434} C_VEL
LIN {X 0,Y 712.025,Z 923.03,A -85,B 0,C 180,E1 2866.501,E2 2866.501} C_VEL
LIN {X 0,Y 712.242,Z 923.03,A -85,B 0,C 180,E1 2870.229,E2 2870.229} C_VEL
LIN {X 0,Y 712.059,Z 923.03,A -85,B 0,C 180,E1 2875.132,E2 2875.132} C_VEL
LIN {X 0,Y 712.217,Z 923.03,A -85,B 0,C 180,E1 2877.151,E2 2877.151} C_VEL
LIN {X 0,Y 713.764,Z 944.574,A -85,B 0,C 180,E1 2877.423,E2 2877.423} C_VEL
LIN {X 0,Y 713.703,Z 974.677,A -85,B 0,C 180,E1 2877.916,E2 2877.916} C_VEL
LIN {X 0,Y 713.366,Z 1003.118,A -85,B 0,C 180,E1 2878.863,E2 2878.863} C_VEL
LIN {X 0,Y 713.106,Z 1028.215,A -85,B 0,C 180,E1 2880.229,E2 2880.229} C_VEL
LIN {X 0,Y 712.852,Z 1049.823,A -85,B 0,C 180,E1 2881.975,E2 2881.975} C_VEL
LIN {X 0,Y 712.717,Z 1066.069,A -85,B 0,C 180,E1 2883.906,E2 2883.906} C_VEL
LIN {X 0,Y 712.584,Z 1077.861,A -85,B 0,C 180,E1 2886.088,E2 2886.088} C_VEL
LIN {X 0,Y 712.529,Z 1083.357,A -85,B 0,C 180,E1 2887.925,E2 2887.925} C_VEL
LIN {X 0,Y 712.493,Z 1085.419,A -85,B 0,C 180,E1 2889.77,E2 2889.77} C_VEL
LIN {X 0,Y 712.537,Z 1082.791,A -85,B 0,C 180,E1 2892.245,E2 2892.245} C_VEL
LIN {X 0,Y 712.6,Z 1075.151,A -85,B 0,C 180,E1 2894.429,E2 2894.429} C_VEL
LIN {X 0,Y 712.775,Z 1061.567,A -85,B 0,C 180,E1 2896.632,E2 2896.632} C_VEL
LIN {X 0,Y 712.961,Z 1043.32,A -85,B 0,C 180,E1 2898.539,E2 2898.539} C_VEL
LIN {X 0,Y 713.151,Z 1020.79,A -85,B 0,C 180,E1 2900.142,E2 2900.142} C_VEL
LIN {X 0,Y 713.464,Z 994.955,A -85,B 0,C 180,E1 2901.368,E2 2901.368} C_VEL
LIN {X 0,Y 713.76,Z 966.181,A -85,B 0,C 180,E1 2902.186,E2 2902.186} C_VEL
LIN {X 0,Y 712.709,Z 926.609,A -85,B 0,C 180,E1 2902.688,E2 2902.688} C_VEL
LIN {X 0,Y 712.196,Z 923.03,A -85,B 0,C 180,E1 2902.781,E2 2902.781} C_VEL
LIN {X 0,Y 711.916,Z 923.03,A -85,B 0,C 180,E1 2907.839,E2 2907.839} C_VEL
LIN {X 0,Y 711.933,Z 923.03,A -85,B 0,C 180,E1 2912.05,E2 2912.05} C_VEL
LIN {X 0,Y 711.912,Z 923.03,A -85,B 0,C 180,E1 2916.466,E2 2916.466} C_VEL
LIN {X 0,Y 711.796,Z 923.03,A -85,B 0,C 180,E1 2921.158,E2 2921.158} C_VEL
LIN {X 0,Y 711.895,Z 923.03,A -85,B 0,C 180,E1 2926.197,E2 2926.197} C_VEL
LIN {X 0,Y 711.974,Z 923.03,A -85,B 0,C 180,E1 2930.443,E2 2930.443} C_VEL
LIN {X 0,Y 711.88,Z 923.03,A -85,B 0,C 180,E1 2935.881,E2 2935.881} C_VEL
LIN {X 0,Y 711.961,Z 923.03,A -85,B 0,C 180,E1 2940.771,E2 2940.771} C_VEL
LIN {X 0,Y 712.099,Z 923.03,A -85,B 0,C 180,E1 2944.878,E2 2944.878} C_VEL
LIN {X 0,Y 712.044,Z 923.03,A -85,B 0,C 180,E1 2950.141,E2 2950.141} C_VEL
LIN {X 0,Y 712.114,Z 923.03,A -85,B 0,C 180,E1 2955.238,E2 2955.238} C_VEL
LIN {X 0,Y 712.234,Z 923.03,A -85,B 0,C 180,E1 2960.218,E2 2960.218} C_VEL
LIN {X 0,Y 712.223,Z 923.03,A -85,B 0,C 180,E1 2965.121,E2 2965.121} C_VEL
LIN {X 0,Y 712.3,Z 923.03,A -85,B 0,C 180,E1 2969.989,E2 2969.989} C_VEL
LIN {X 0,Y 712.437,Z 923.03,A -85,B 0,C 180,E1 2974.856,E2 2974.856} C_VEL
LIN {X 0,Y 712.185,Z 923.03,A -85,B 0,C 180,E1 2979.761,E2 2979.761} C_VEL
LIN {X 0,Y 712.138,Z 923.03,A -85,B 0,C 180,E1 2984.739,E2 2984.739} C_VEL
LIN {X 0,Y 712.139,Z 923.03,A -85,B 0,C 180,E1 2988.546,E2 2988.546} C_VEL
LIN {X 0,Y 712.078,Z 923.03,A -85,B 0,C 180,E1 2993.764,E2 2993.764} C_VEL
LIN {X 0,Y 712.015,Z 923.03,A -85,B 0,C 180,E1 2999.202,E2 2999.202} C_VEL
LIN {X 0,Y 711.988,Z 923.03,A -85,B 0,C 180,E1 3004.132,E2 3004.132} C_VEL
LIN {X 0,Y 711.875,Z 923.03,A -85,B 0,C 180,E1 3008.24,E2 3008.24} C_VEL
LIN {X 0,Y 712.196,Z 923.03,A -85,B 0,C 180,E1 3013.829,E2 3013.829} C_VEL
LIN {X 0,Y 711.884,Z 923.03,A -85,B 0,C 180,E1 3018.849,E2 3018.849} C_VEL
LIN {X 0,Y 711.922,Z 923.03,A -85,B 0,C 180,E1 3023.737,E2 3023.737} C_VEL
LIN {X 0,Y 711.972,Z 923.03,A -85,B 0,C 180,E1 3029.376,E2 3029.376} C_VEL
LIN {X 0,Y 712.195,Z 923.03,A -85,B 0,C 180,E1 3034.889,E2 3034.889} C_VEL
LIN {X 0,Y 712.271,Z 923.03,A -85,B 0,C 180,E1 3035.648,E2 3035.648} C_VEL
LIN {X 0,Y 716.607,Z 939.586,A -85,B 0,C 180,E1 3036.065,E2 3036.065} C_VEL
LIN {X 0,Y 716.137,Z 981.525,A -85,B 0,C 180,E1 3037.097,E2 3037.097} C_VEL
LIN {X 0,Y 715.339,Z 1019.05,A -85,B 0,C 180,E1 3038.53,E2 3038.53} C_VEL
LIN {X 0,Y 714.491,Z 1055.187,A -85,B 0,C 180,E1 3040.461,E2 3040.461} C_VEL
LIN {X 0,Y 713.812,Z 1087.214,A -85,B 0,C 180,E1 3042.759,E2 3042.759} C_VEL
LIN {X 0,Y 713.228,Z 1115.396,A -85,B 0,C 180,E1 3045.427,E2 3045.427} C_VEL
LIN {X 0,Y 712.827,Z 1138.721,A -85,B 0,C 180,E1 3048.381,E2 3048.381} C_VEL
LIN {X 0,Y 712.579,Z 1156.187,A -85,B 0,C 180,E1 3051.462,E2 3051.462} C_VEL
LIN {X 0,Y 712.48,Z 1167.713,A -85,B 0,C 180,E1 3054.522,E2 3054.522} C_VEL
LIN {X 0,Y 712.427,Z 1173.967,A -85,B 0,C 180,E1 3057.567,E2 3057.567} C_VEL
LIN {X 0,Y 712.289,Z 1175.495,A -85,B 0,C 180,E1 3059.999,E2 3059.999} C_VEL
LIN {X 0,Y 712.457,Z 1173.844,A -85,B 0,C 180,E1 3062.43,E2 3062.43} C_VEL
LIN {X 0,Y 712.485,Z 1167.438,A -85,B 0,C 180,E1 3065.475,E2 3065.475} C_VEL
LIN {X 0,Y 712.54,Z 1155.777,A -85,B 0,C 180,E1 3068.536,E2 3068.536} C_VEL
LIN {X 0,Y 712.762,Z 1140.262,A -85,B 0,C 180,E1 3071.291,E2 3071.291} C_VEL
LIN {X 0,Y 709.001,Z 1132.363,A -85,B 0,C 180,E1 3072.517,E2 3072.517} C_VEL
LIN {X 0,Y 705.251,Z 1123.5,A -85,B 0,C 180,E1 3073.709,E2 3073.709} C_VEL
LIN {X 0,Y 705.88,Z 1097.163,A -85,B 0,C 180,E1 3076.477,E2 3076.477} C_VEL
LIN {X 0,Y 706.711,Z 1066.18,A -85,B 0,C 180,E1 3078.939,E2 3078.939} C_VEL
LIN {X 0,Y 707.612,Z 1032.514,A -85,B 0,C 180,E1 3080.957,E2 3080.957} C_VEL
LIN {X 0,Y 708.48,Z 995.756,A -85,B 0,C 180,E1 3082.575,E2 3082.575} C_VEL
LIN {X 0,Y 709.302,Z 956.565,A -85,B 0,C 180,E1 3083.747,E2 3083.747} C_VEL
LIN {X 0,Y 708.598,Z 936.464,A -85,B 0,C 180,E1 3084.186,E2 3084.186} C_VEL
LIN {X 0,Y 704.135,Z 923.03,A -85,B 0,C 180,E1 3084.59,E2 3084.59} C_VEL
LIN {X 0,Y 704.101,Z 923.03,A -85,B 0,C 180,E1 3089.577,E2 3089.577} C_VEL
LIN {X 0,Y 704.093,Z 923.03,A -85,B 0,C 180,E1 3093.916,E2 3093.916} C_VEL
LIN {X 0,Y 703.934,Z 923.03,A -85,B 0,C 180,E1 3098.499,E2 3098.499} C_VEL
LIN {X 0,Y 703.969,Z 923.03,A -85,B 0,C 180,E1 3103.383,E2 3103.383} C_VEL
LIN {X 0,Y 703.948,Z 923.03,A -85,B 0,C 180,E1 3108.702,E2 3108.702} C_VEL
LIN {X 0,Y 704.059,Z 923.03,A -85,B 0,C 180,E1 3113.079,E2 3113.079} C_VEL
LIN {X 0,Y 704.04,Z 923.03,A -85,B 0,C 180,E1 3117.565,E2 3117.565} C_VEL
LIN {X 0,Y 704.019,Z 923.03,A -85,B 0,C 180,E1 3121.838,E2 3121.838} C_VEL
LIN {X 0,Y 703.929,Z 923.03,A -85,B 0,C 180,E1 3124.694,E2 3124.694} C_VEL
LIN {X 0,Y 709.818,Z 941.214,A -85,B 0,C 180,E1 3125.136,E2 3125.136} C_VEL
LIN {X 0,Y 709.52,Z 1001.198,A -85,B 0,C 180,E1 3125.884,E2 3125.884} C_VEL
LIN {X 0,Y 708.834,Z 1042.053,A -85,B 0,C 180,E1 3126.91,E2 3126.91} C_VEL
LIN {X 0,Y 707.92,Z 1080.714,A -85,B 0,C 180,E1 3128.419,E2 3128.419} C_VEL
LIN {X 0,Y 706.979,Z 1115.55,A -85,B 0,C 180,E1 3130.316,E2 3130.316} C_VEL
LIN {X 0,Y 706.058,Z 1146.81,A -85,B 0,C 180,E1 3132.578,E2 3132.578} C_VEL
LIN {X 0,Y 705.399,Z 1173.628,A -85,B 0,C 180,E1 3135.117,E2 3135.117} C_VEL
LIN {X 0,Y 704.987,Z 1196.319,A -85,B 0,C 180,E1 3137.949,E2 3137.949} C_VEL
LIN {X 0,Y 704.707,Z 1213.963,A -85,B 0,C 180,E1 3140.957,E2 3140.957} C_VEL
LIN {X 0,Y 704.574,Z 1225.691,A -85,B 0,C 180,E1 3143.856,E2 3143.856} C_VEL
LIN {X 0,Y 704.489,Z 1231.97,A -85,B 0,C 180,E1 3146.322,E2 3146.322} C_VEL
LIN {X 0,Y 704.499,Z 1235.094,A -85,B 0,C 180,E1 3148.782,E2 3148.782} C_VEL
LIN {X 0,Y 704.635,Z 1235.077,A -85,B 0,C 180,E1 3151.24,E2 3151.24} C_VEL
LIN {X 0,Y 704.586,Z 1230.584,A -85,B 0,C 180,E1 3154.373,E2 3154.373} C_VEL
LIN {X 0,Y 704.694,Z 1219.976,A -85,B 0,C 180,E1 3157.712,E2 3157.712} C_VEL
LIN {X 0,Y 704.838,Z 1204.282,A -85,B 0,C 180,E1 3160.822,E2 3160.822} C_VEL
LIN {X 0,Y 705.245,Z 1183.095,A -85,B 0,C 180,E1 3163.8,E2 3163.8} C_VEL
LIN {X 0,Y 705.819,Z 1157.495,A -85,B 0,C 180,E1 3166.489,E2 3166.489} C_VEL
LIN {X 0,Y 706.601,Z 1127.857,A -85,B 0,C 180,E1 3168.867,E2 3168.867} C_VEL
LIN {X 0,Y 707.558,Z 1094.674,A -85,B 0,C 180,E1 3170.888,E2 3170.888} C_VEL
LIN {X 0,Y 708.449,Z 1058.808,A -85,B 0,C 180,E1 3172.503,E2 3172.503} C_VEL
LIN {X 0,Y 709.259,Z 1021.448,A -85,B 0,C 180,E1 3173.669,E2 3173.669} C_VEL
LIN {X 0,Y 709.703,Z 984.456,A -85,B 0,C 180,E1 3174.378,E2 3174.378} C_VEL
LIN {X 0,Y 709.167,Z 937.805,A -85,B 0,C 180,E1 3174.926,E2 3174.926} C_VEL
LIN {X 0,Y 703.965,Z 923.03,A -85,B 0,C 180,E1 3175.328,E2 3175.328} C_VEL
LIN {X 0,Y 704.101,Z 923.03,A -85,B 0,C 180,E1 3179.588,E2 3179.588} C_VEL
LIN {X 0,Y 704.105,Z 923.03,A -85,B 0,C 180,E1 3183.926,E2 3183.926} C_VEL
LIN {X 0,Y 703.923,Z 923.03,A -85,B 0,C 180,E1 3188.511,E2 3188.511} C_VEL
LIN {X 0,Y 703.977,Z 923.03,A -85,B 0,C 180,E1 3193.394,E2 3193.394} C_VEL
LIN {X 0,Y 703.953,Z 923.03,A -85,B 0,C 180,E1 3198.714,E2 3198.714} C_VEL
LIN {X 0,Y 704.06,Z 923.03,A -85,B 0,C 180,E1 3203.063,E2 3203.063} C_VEL
LIN {X 0,Y 703.995,Z 923.03,A -85,B 0,C 180,E1 3207.548,E2 3207.548} C_VEL
LIN {X 0,Y 704.072,Z 923.03,A -85,B 0,C 180,E1 3211.826,E2 3211.826} C_VEL
LIN {X 0,Y 704.207,Z 923.03,A -85,B 0,C 180,E1 3215.941,E2 3215.941} C_VEL
LIN {X 0,Y 704.007,Z 923.03,A -85,B 0,C 180,E1 3220.826,E2 3220.826} C_VEL
LIN {X 0,Y 704.113,Z 923.03,A -85,B 0,C 180,E1 3226.347,E2 3226.347} C_VEL
LIN {X 0,Y 704.255,Z 923.03,A -85,B 0,C 180,E1 3230.788,E2 3230.788} C_VEL
LIN {X 0,Y 704.161,Z 923.03,A -85,B 0,C 180,E1 3235.077,E2 3235.077} C_VEL
LIN {X 0,Y 704.306,Z 923.03,A -85,B 0,C 180,E1 3237.019,E2 3237.019} C_VEL
LIN {X 0,Y 706.051,Z 944.539,A -85,B 0,C 180,E1 3237.287,E2 3237.287} C_VEL
LIN {X 0,Y 705.98,Z 974.53,A -85,B 0,C 180,E1 3237.778,E2 3237.778} C_VEL
LIN {X 0,Y 705.646,Z 1002.211,A -85,B 0,C 180,E1 3238.698,E2 3238.698} C_VEL
LIN {X 0,Y 705.263,Z 1027.599,A -85,B 0,C 180,E1 3240.078,E2 3240.078} C_VEL
LIN {X 0,Y 704.996,Z 1049.38,A -85,B 0,C 180,E1 3241.844,E2 3241.844} C_VEL
LIN {X 0,Y 704.839,Z 1066.433,A -85,B 0,C 180,E1 3243.892,E2 3243.892} C_VEL
LIN {X 0,Y 704.686,Z 1078.324,A -85,B 0,C 180,E1 3246.156,E2 3246.156} C_VEL
LIN {X 0,Y 704.625,Z 1083.583,A -85,B 0,C 180,E1 3248.014,E2 3248.014} C_VEL
LIN {X 0,Y 704.592,Z 1085.404,A -85,B 0,C 180,E1 3249.881,E2 3249.881} C_VEL
LIN {X 0,Y 704.655,Z 1082.53,A -85,B 0,C 180,E1 3252.384,E2 3252.384} C_VEL
LIN {X 0,Y 704.722,Z 1074.626,A -85,B 0,C 180,E1 3254.594,E2 3254.594} C_VEL
LIN {X 0,Y 704.881,Z 1060.652,A -85,B 0,C 180,E1 3256.824,E2 3256.824} C_VEL
LIN {X 0,Y 705.13,Z 1041.898,A -85,B 0,C 180,E1 3258.752,E2 3258.752} C_VEL
LIN {X 0,Y 705.366,Z 1018.733,A -85,B 0,C 180,E1 3260.374,E2 3260.374} C_VEL
LIN {X 0,Y 705.734,Z 992.741,A -85,B 0,C 180,E1 3261.585,E2 3261.585} C_VEL
LIN {X 0,Y 706.035,Z 963.679,A -85,B 0,C 180,E1 3262.37,E2 3262.37} C_VEL
LIN {X 0,Y 705.007,Z 927.542,A -85,B 0,C 180,E1 3262.816,E2 3262.816} C_VEL
LIN {X 0,Y 704.283,Z 923.03,A -85,B 0,C 180,E1 3262.904,E2 3262.904} C_VEL
LIN {X 0,Y 703.971,Z 923.03,A -85,B 0,C 180,E1 3268.181,E2 3268.181} C_VEL
LIN {X 0,Y 703.972,Z 923.03,A -85,B 0,C 180,E1 3273.148,E2 3273.148} C_VEL
LIN {X 0,Y 704.012,Z 923.03,A -85,B 0,C 180,E1 3278.498,E2 3278.498} C_VEL
LIN {X 0,Y 703.847,Z 923.03,A -85,B 0,C 180,E1 3283.396,E2 3283.396} C_VEL
LIN {X 0,Y 703.997,Z 923.03,A -85,B 0,C 180,E1 3288.702,E2 3288.702} C_VEL
LIN {X 0,Y 703.931,Z 923.03,A -85,B 0,C 180,E1 3293.044,E2 3293.044} C_VEL
LIN {X 0,Y 703.937,Z 923.03,A -85,B 0,C 180,E1 3297.534,E2 3297.534} C_VEL
LIN {X 0,Y 704.11,Z 923.03,A -85,B 0,C 180,E1 3301.817,E2 3301.817} C_VEL
LIN {X 0,Y 704.156,Z 923.03,A -85,B 0,C 180,E1 3305.928,E2 3305.928} C_VEL
LIN {X 0,Y 704.213,Z 923.03,A -85,B 0,C 180,E1 3311.214,E2 3311.214} C_VEL
LIN {X 0,Y 704.101,Z 923.03,A -85,B 0,C 180,E1 3316.335,E2 3316.335} C_VEL
LIN {X 0,Y 704.241,Z 923.03,A -85,B 0,C 180,E1 3321.351,E2 3321.351} C_VEL
LIN {X 0,Y 704.436,Z 923.03,A -85,B 0,C 180,E1 3326.3,E2 3326.3} C_VEL
LIN {X 0,Y 704.569,Z 923.03,A -85,B 0,C 180,E1 3331.218,E2 3331.218} C_VEL
LIN {X 0,Y 704.329,Z 923.03,A -85,B 0,C 180,E1 3336.147,E2 3336.147} C_VEL
LIN {X 0,Y 704.242,Z 923.03,A -85,B 0,C 180,E1 3341.122,E2 3341.122} C_VEL
LIN {X 0,Y 704.307,Z 923.03,A -85,B 0,C 180,E1 3346.183,E2 3346.183} C_VEL
LIN {X 0,Y 704.157,Z 923.03,A -85,B 0,C 180,E1 3351.382,E2 3351.382} C_VEL
LIN {X 0,Y 704.15,Z 923.03,A -85,B 0,C 180,E1 3355.666,E2 3355.666} C_VEL
LIN {X 0,Y 704.106,Z 923.03,A -85,B 0,C 180,E1 3360.986,E2 3360.986} C_VEL
LIN {X 0,Y 704.042,Z 923.03,A -85,B 0,C 180,E1 3365.399,E2 3365.399} C_VEL
LIN {X 0,Y 703.906,Z 923.03,A -85,B 0,C 180,E1 3370.074,E2 3370.074} C_VEL
LIN {X 0,Y 704.195,Z 923.03,A -85,B 0,C 180,E1 3374.915,E2 3374.915} C_VEL
LIN {X 0,Y 704.03,Z 923.03,A -85,B 0,C 180,E1 3380.572,E2 3380.572} C_VEL
LIN {X 0,Y 703.971,Z 923.03,A -85,B 0,C 180,E1 3386.074,E2 3386.074} C_VEL
LIN {X 0,Y 704.051,Z 923.03,A -85,B 0,C 180,E1 3390.418,E2 3390.418} C_VEL
LIN {X 0,Y 704.341,Z 923.181,A -85,B 0,C 180,E1 3395.362,E2 3395.362} C_VEL
LIN {X 0,Y 709.38,Z 940.901,A -85,B 0,C 180,E1 3395.828,E2 3395.828} C_VEL
LIN {X 0,Y 708.781,Z 982.454,A -85,B 0,C 180,E1 3396.878,E2 3396.878} C_VEL
LIN {X 0,Y 707.899,Z 1019.881,A -85,B 0,C 180,E1 3398.334,E2 3398.334} C_VEL
LIN {X 0,Y 706.924,Z 1054.71,A -85,B 0,C 180,E1 3400.214,E2 3400.214} C_VEL
LIN {X 0,Y 706.096,Z 1087.212,A -85,B 0,C 180,E1 3402.564,E2 3402.564} C_VEL
LIN {X 0,Y 705.461,Z 1115.394,A -85,B 0,C 180,E1 3405.263,E2 3405.263} C_VEL
LIN {X 0,Y 704.955,Z 1138.718,A -85,B 0,C 180,E1 3408.249,E2 3408.249} C_VEL
LIN {X 0,Y 704.691,Z 1156.183,A -85,B 0,C 180,E1 3411.366,E2 3411.366} C_VEL
LIN {X 0,Y 704.572,Z 1167.713,A -85,B 0,C 180,E1 3414.46,E2 3414.46} C_VEL
LIN {X 0,Y 704.531,Z 1173.967,A -85,B 0,C 180,E1 3417.54,E2 3417.54} C_VEL
LIN {X 0,Y 704.39,Z 1175.495,A -85,B 0,C 180,E1 3419.999,E2 3419.999} C_VEL
LIN {X 0,Y 704.559,Z 1173.846,A -85,B 0,C 180,E1 3422.457,E2 3422.457} C_VEL
LIN {X 0,Y 704.584,Z 1167.441,A -85,B 0,C 180,E1 3425.537,E2 3425.537} C_VEL
LIN {X 0,Y 704.651,Z 1155.781,A -85,B 0,C 180,E1 3428.632,E2 3428.632} C_VEL
LIN {X 0,Y 704.93,Z 1138.117,A -85,B 0,C 180,E1 3431.749,E2 3431.749} C_VEL
LIN {X 0,Y 705.251,Z 1123.5,A -85,B 0,C 180,E1 3433.709,E2 3433.709} C_VEL
LIN {X 0,Y 701.509,Z 1114.077,A -85,B 0,C 180,E1 3434.875,E2 3434.875} C_VEL
LIN {X 0,Y 697.968,Z 1103.957,A -85,B 0,C 180,E1 3436.014,E2 3436.014} C_VEL
LIN {X 0,Y 698.819,Z 1075.331,A -85,B 0,C 180,E1 3438.489,E2 3438.489} C_VEL
LIN {X 0,Y 699.836,Z 1041.531,A -85,B 0,C 180,E1 3440.704,E2 3440.704} C_VEL
LIN {X 0,Y 700.938,Z 1003.795,A -85,B 0,C 180,E1 3442.518,E2 3442.518} C_VEL
LIN {X 0,Y 701.873,Z 964.175,A -85,B 0,C 180,E1 3443.82,E2 3443.82} C_VEL
LIN {X 0,Y 701.65,Z 939.238,A -85,B 0,C 180,E1 3444.394,E2 3444.394} C_VEL
LIN {X 0,Y 696.191,Z 923.03,A -85,B 0,C 180,E1 3444.875,E2 3444.875} C_VEL
LIN {X 0,Y 696.173,Z 923.03,A -85,B 0,C 180,E1 3449.948,E2 3449.948} C_VEL
LIN {X 0,Y 696.12,Z 923.03,A -85,B 0,C 180,E1 3454.451,E2 3454.451} C_VEL
LIN {X 0,Y 695.983,Z 923.03,A -85,B 0,C 180,E1 3459.022,E2 3459.022} C_VEL
LIN {X 0,Y 695.959,Z 923.03,A -85,B 0,C 180,E1 3464.254,E2 3464.254} C_VEL
LIN {X 0,Y 695.987,Z 923.03,A -85,B 0,C 180,E1 3469.454,E2 3469.454} C_VEL
LIN {X 0,Y 696.161,Z 923.03,A -85,B 0,C 180,E1 3474.139,E2 3474.139} C_VEL
LIN {X 0,Y 696.057,Z 923.03,A -85,B 0,C 180,E1 3478.615,E2 3478.615} C_VEL
LIN {X 0,Y 696.023,Z 923.03,A -85,B 0,C 180,E1 3482.891,E2 3482.891} C_VEL
LIN {X 0,Y 696.002,Z 923.126,A -85,B 0,C 180,E1 3484.405,E2 3484.405} C_VEL
LIN {X 0,Y 702.601,Z 941.357,A -85,B 0,C 180,E1 3484.864,E2 3484.864} C_VEL
LIN {X 0,Y 702.298,Z 1001.749,A -85,B 0,C 180,E1 3485.63,E2 3485.63} C_VEL
LIN {X 0,Y 701.524,Z 1041.518,A -85,B 0,C 180,E1 3486.637,E2 3486.637} C_VEL
LIN {X 0,Y 700.518,Z 1079.525,A -85,B 0,C 180,E1 3488.121,E2 3488.121} C_VEL
LIN {X 0,Y 699.427,Z 1115.342,A -85,B 0,C 180,E1 3490.081,E2 3490.081} C_VEL
LIN {X 0,Y 698.413,Z 1146.809,A -85,B 0,C 180,E1 3492.381,E2 3492.381} C_VEL
LIN {X 0,Y 697.651,Z 1173.627,A -85,B 0,C 180,E1 3494.948,E2 3494.948} C_VEL
LIN {X 0,Y 697.129,Z 1196.317,A -85,B 0,C 180,E1 3497.811,E2 3497.811} C_VEL
LIN {X 0,Y 696.844,Z 1213.963,A -85,B 0,C 180,E1 3500.854,E2 3500.854} C_VEL
LIN {X 0,Y 696.685,Z 1225.691,A -85,B 0,C 180,E1 3503.786,E2 3503.786} C_VEL
LIN {X 0,Y 696.606,Z 1231.97,A -85,B 0,C 180,E1 3506.28,E2 3506.28} C_VEL
LIN {X 0,Y 696.599,Z 1235.095,A -85,B 0,C 180,E1 3508.768,E2 3508.768} C_VEL
LIN {X 0,Y 696.733,Z 1235.077,A -85,B 0,C 180,E1 3511.254,E2 3511.254} C_VEL
LIN {X 0,Y 696.7,Z 1230.848,A -85,B 0,C 180,E1 3514.302,E2 3514.302} C_VEL
LIN {X 0,Y 696.742,Z 1221.231,A -85,B 0,C 180,E1 3517.487,E2 3517.487} C_VEL
LIN {X 0,Y 696.941,Z 1206.149,A -85,B 0,C 180,E1 3520.63,E2 3520.63} C_VEL
LIN {X 0,Y 697.417,Z 1184.417,A -85,B 0,C 180,E1 3523.798,E2 3523.798} C_VEL
LIN {X 0,Y 698.076,Z 1159.246,A -85,B 0,C 180,E1 3526.516,E2 3526.516} C_VEL
LIN {X 0,Y 698.993,Z 1129.939,A -85,B 0,C 180,E1 3528.931,E2 3528.931} C_VEL
LIN {X 0,Y 700.03,Z 1096.202,A -85,B 0,C 180,E1 3531.04,E2 3531.04} C_VEL
LIN {X 0,Y 701.052,Z 1060.353,A -85,B 0,C 180,E1 3532.693,E2 3532.693} C_VEL
LIN {X 0,Y 701.965,Z 1022.935,A -85,B 0,C 180,E1 3533.892,E2 3533.892} C_VEL
LIN {X 0,Y 702.521,Z 984.552,A -85,B 0,C 180,E1 3534.643,E2 3534.643} C_VEL
LIN {X 0,Y 701.886,Z 939.599,A -85,B 0,C 180,E1 3535.182,E2 3535.182} C_VEL
LIN {X 0,Y 696.017,Z 923.03,A -85,B 0,C 180,E1 3535.652,E2 3535.652} C_VEL
LIN {X 0,Y 696.167,Z 923.03,A -85,B 0,C 180,E1 3539.959,E2 3539.959} C_VEL
LIN {X 0,Y 696.136,Z 923.03,A -85,B 0,C 180,E1 3544.428,E2 3544.428} C_VEL
LIN {X 0,Y 695.985,Z 923.03,A -85,B 0,C 180,E1 3549.033,E2 3549.033} C_VEL
LIN {X 0,Y 695.99,Z 923.03,A -85,B 0,C 180,E1 3554.237,E2 3554.237} C_VEL
LIN {X 0,Y 695.994,Z 923.03,A -85,B 0,C 180,E1 3559.466,E2 3559.466} C_VEL
LIN {X 0,Y 696.141,Z 923.03,A -85,B 0,C 180,E1 3564.122,E2 3564.122} C_VEL
LIN {X 0,Y 696.035,Z 923.03,A -85,B 0,C 180,E1 3568.599,E2 3568.599} C_VEL
LIN {X 0,Y 696.149,Z 923.03,A -85,B 0,C 180,E1 3572.883,E2 3572.883} C_VEL
LIN {X 0,Y 696.218,Z 923.03,A -85,B 0,C 180,E1 3577.005,E2 3577.005} C_VEL
LIN {X 0,Y 696.1,Z 923.03,A -85,B 0,C 180,E1 3580.998,E2 3580.998} C_VEL
LIN {X 0,Y 696.195,Z 923.03,A -85,B 0,C 180,E1 3586.188,E2 3586.188} C_VEL
LIN {X 0,Y 696.349,Z 923.03,A -85,B 0,C 180,E1 3591.264,E2 3591.264} C_VEL
LIN {X 0,Y 696.283,Z 923.03,A -85,B 0,C 180,E1 3596.268,E2 3596.268} C_VEL
LIN {X 0,Y 696.385,Z 923.319,A -85,B 0,C 180,E1 3596.899,E2 3596.899} C_VEL
LIN {X 0,Y 698.33,Z 943.996,A -85,B 0,C 180,E1 3597.149,E2 3597.149} C_VEL
LIN {X 0,Y 698.274,Z 974.529,A -85,B 0,C 180,E1 3597.637,E2 3597.637} C_VEL
LIN {X 0,Y 697.918,Z 1001.74,A -85,B 0,C 180,E1 3598.528,E2 3598.528} C_VEL
LIN {X 0,Y 697.537,Z 1026.51,A -85,B 0,C 180,E1 3599.846,E2 3599.846} C_VEL
LIN {X 0,Y 697.227,Z 1047.866,A -85,B 0,C 180,E1 3601.554,E2 3601.554} C_VEL
LIN {X 0,Y 696.993,Z 1064.904,A -85,B 0,C 180,E1 3603.575,E2 3603.575} C_VEL
LIN {X 0,Y 696.782,Z 1077.47,A -85,B 0,C 180,E1 3605.914,E2 3605.914} C_VEL
LIN {X 0,Y 696.732,Z 1083.809,A -85,B 0,C 180,E1 3608.106,E2 3608.106} C_VEL
LIN {X 0,Y 696.678,Z 1085.388,A -85,B 0,C 180,E1 3609.994,E2 3609.994} C_VEL
LIN {X 0,Y 696.781,Z 1082.163,A -85,B 0,C 180,E1 3612.576,E2 3612.576} C_VEL
